KUKA KRL program: EPS_2_25730_SANMH01_A_20250909085214.src

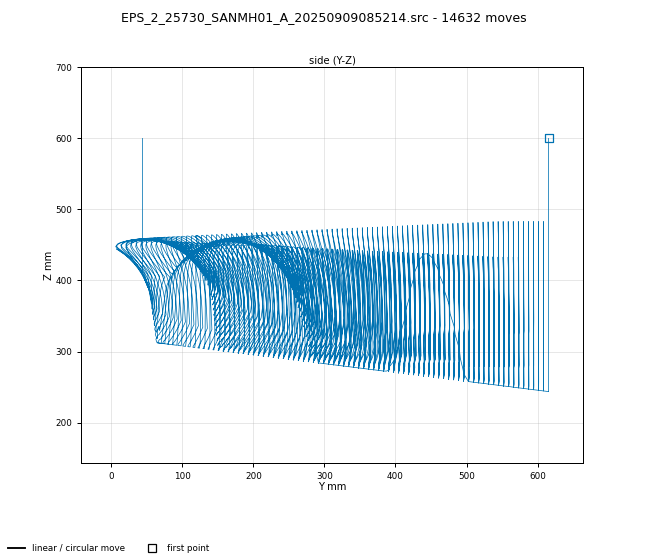
[picture p0: tool path of EPS_2_25730_SANMH01_A_20250909085214.src, 14632 of 14634 moves have a stored position in this frame; points joined in program order, loops and branches not executed]
&ACCESS RVP
&REL 4
&COMMENT QRS 19112012
&PARAM EDITMASK = *
DEF PART()
EXT BAS (BAS_COMMAND :IN,REAL :IN )
INT I
BAS (#INITMOV,0 )

;KUKA QRS Post kuka4.cps  Date:22-06-2017 !

File_ID=2821

QRS_PRE_INIT()

;Init var - Until changes are made in qrs_pre_init
Outlet_Square_prg=0
Inlet_1_Square_prg=0
Inlet_2_Square_prg=0
Inlet_3_Square_prg=0
Inlet_4_Square_prg=0
Inlet_5_Square_prg=0

Outlet_1={X 0.000, Y 541.230, Z 408.000, B 0.000, E1 0.000 }
Inlet_1={X 0.000, Y 544.780, Z 358.000, B 0.000, E1 163.000 }
Inlet_2={X 0.000, Y 544.780, Z 358.000, B 0.000, E1 270.000 }
Outlet_1_type=150
Inlet_1_type=150
Inlet_2_type=150
;QRS#1=Sidecore dimensions
;QRS#2=150-6" PVC SDR 28
;QRS#3=150-6" PVC SDR 28
;QRS#4=150-6" PVC SDR 28
;QRS#5=
;QRS#6=
;QRS#7=
;QRS#8=
;QRS#9=10-06 PSX
;QRS#10=10-06 PSX
;QRS#11=10-06 PSX
;QRS#12=
;QRS#13=
;QRS#14=
;QRS#15=
;QRS#16=1220x127x762 2,5'
;QRS#17=EPS Height
;QRS#18=483
;QRS#19=*
;QRS#20= UPDATED VERSION 22-06-2017
;QRS#21=*
Outlet_Square=070
Inlet_1_Square=070
Inlet_2_Square=070
Inlet_3_Square=0
Inlet_4_Square=0
Inlet_5_Square=0
Mill_Square=1
Outlet_Square_Prg=203
Inlet_1_Square_prg=203
Inlet_2_Square_prg=203

QRS_INIT()

$ADVANCE=5

; T1
PTP {E1 173.628,E2 173.628}
PTP {X 0,Y 615.477,A -85,B 0,C 180,E1 173.628,E2 173.628,E3 0,E4 0,E5 0,E6 0}
QRS_SPEED_INIT()
LIN {X 0,Y 615.477,Z 600,A -85,B 0,C 180,E1 173.628,E2 173.628,E3 0,E4 0,E5 0,E6 0} C_VEL
LIN {X 0,Y 615.477,Z 253.689,A -85,B 0,C 180,E1 173.628,E2 173.628} C_VEL
LIN {X 0,Y 615.477,Z 245.508,A -85,B 0,C 180,E1 173.628,E2 173.628} C_VEL
LIN {X 0,Y 615.462,Z 243.508,A -85,B 0,C 180,E1 173.442,E2 173.442} C_VEL
LIN {X 0,Y 615.457,Z 243.501,A -85,B 0,C 180,E1 170.803,E2 170.803} C_VEL
LIN {X 0,Y 615.49,Z 243.501,A -85,B 0,C 180,E1 168.142,E2 168.142} C_VEL
LIN {X 0,Y 615.471,Z 243.51,A -85,B 0,C 180,E1 165.453,E2 165.453} C_VEL
LIN {X 0,Y 615.469,Z 243.509,A -85,B 0,C 180,E1 163.416,E2 163.416} C_VEL
LIN {X 0,Y 615.466,Z 243.509,A -85,B 0,C 180,E1 161.356,E2 161.356} C_VEL
LIN {X 0,Y 615.462,Z 243.509,A -85,B 0,C 180,E1 159.271,E2 159.271} C_VEL
LIN {X 0,Y 615.456,Z 243.508,A -85,B 0,C 180,E1 157.157,E2 157.157} C_VEL
LIN {X 0,Y 615.45,Z 243.506,A -85,B 0,C 180,E1 155.01,E2 155.01} C_VEL
LIN {X 0,Y 615.446,Z 243.505,A -85,B 0,C 180,E1 152.824,E2 152.824} C_VEL
LIN {X 0,Y 615.475,Z 243.499,A -85,B 0,C 180,E1 150.207,E2 150.207} C_VEL
LIN {X 0,Y 615.493,Z 243.511,A -85,B 0,C 180,E1 147.547,E2 147.547} C_VEL
LIN {X 0,Y 615.469,Z 243.51,A -85,B 0,C 180,E1 145.188,E2 145.188} C_VEL
LIN {X 0,Y 615.444,Z 243.506,A -85,B 0,C 180,E1 142.759,E2 142.759} C_VEL
LIN {X 0,Y 615.489,Z 243.498,A -85,B 0,C 180,E1 139.911,E2 139.911} C_VEL
LIN {X 0,Y 615.458,Z 243.509,A -85,B 0,C 180,E1 136.956,E2 136.956} C_VEL
LIN {X 0,Y 615.458,Z 243.509,A -85,B 0,C 180,E1 134.934,E2 134.934} C_VEL
LIN {X 0,Y 615.443,Z 243.504,A -85,B 0,C 180,E1 132.357,E2 132.357} C_VEL
LIN {X 0,Y 615.488,Z 243.499,A -85,B 0,C 180,E1 129.75,E2 129.75} C_VEL
LIN {X 0,Y 615.467,Z 243.51,A -85,B 0,C 180,E1 126.94,E2 126.94} C_VEL
LIN {X 0,Y 615.45,Z 243.508,A -85,B 0,C 180,E1 124.702,E2 124.702} C_VEL
LIN {X 0,Y 615.49,Z 243.609,A -85,B 0,C 180,E1 123.602,E2 123.602} C_VEL
LIN {X 0,Y 615.443,Z 256.214,A -85,B 0,C 180,E1 120.922,E2 120.922} C_VEL
LIN {X 0,Y 615.478,Z 267.899,A -85,B 0,C 180,E1 118.457,E2 118.457} C_VEL
LIN {X 0,Y 615.482,Z 274.607,A -85,B 0,C 180,E1 117.053,E2 117.053} C_VEL
LIN {X 0,Y 615.469,Z 350.299,A -85,B 0,C 180,E1 116.148,E2 116.148} C_VEL
LIN {X 0,Y 615.466,Z 359.834,A -85,B 0,C 180,E1 115.944,E2 115.944} C_VEL
LIN {X 0,Y 615.476,Z 369.268,A -85,B 0,C 180,E1 115.647,E2 115.647} C_VEL
LIN {X 0,Y 615.495,Z 380.853,A -85,B 0,C 180,E1 115.137,E2 115.137} C_VEL
LIN {X 0,Y 615.481,Z 389.489,A -85,B 0,C 180,E1 114.632,E2 114.632} C_VEL
LIN {X 0,Y 615.487,Z 396.326,A -85,B 0,C 180,E1 114.145,E2 114.145} C_VEL
LIN {X 0,Y 615.497,Z 403.192,A -85,B 0,C 180,E1 113.556,E2 113.556} C_VEL
LIN {X 0,Y 615.495,Z 410.002,A -85,B 0,C 180,E1 112.844,E2 112.844} C_VEL
LIN {X 0,Y 615.496,Z 416.819,A -85,B 0,C 180,E1 111.96,E2 111.96} C_VEL
LIN {X 0,Y 615.497,Z 422.135,A -85,B 0,C 180,E1 111.08,E2 111.08} C_VEL
LIN {X 0,Y 615.492,Z 426.762,A -85,B 0,C 180,E1 110.033,E2 110.033} C_VEL
LIN {X 0,Y 615.495,Z 429.072,A -85,B 0,C 180,E1 109.338,E2 109.338} C_VEL
LIN {X 0,Y 615.489,Z 430.797,A -85,B 0,C 180,E1 108.618,E2 108.618} C_VEL
LIN {X 0,Y 615.489,Z 431.768,A -85,B 0,C 180,E1 107.957,E2 107.957} C_VEL
LIN {X 0,Y 615.498,Z 432.261,A -85,B 0,C 180,E1 107.27,E2 107.27} C_VEL
LIN {X 0,Y 615.494,Z 432.172,A -85,B 0,C 180,E1 106.448,E2 106.448} C_VEL
LIN {X 0,Y 615.492,Z 431.698,A -85,B 0,C 180,E1 105.905,E2 105.905} C_VEL
LIN {X 0,Y 615.496,Z 430.652,A -85,B 0,C 180,E1 105.226,E2 105.226} C_VEL
LIN {X 0,Y 615.495,Z 429.013,A -85,B 0,C 180,E1 104.549,E2 104.549} C_VEL
LIN {X 0,Y 615.49,Z 425.444,A -85,B 0,C 180,E1 103.537,E2 103.537} C_VEL
LIN {X 0,Y 615.495,Z 422.326,A -85,B 0,C 180,E1 102.865,E2 102.865} C_VEL
LIN {X 0,Y 615.495,Z 417.37,A -85,B 0,C 180,E1 102.028,E2 102.028} C_VEL
LIN {X 0,Y 615.5,Z 411.091,A -85,B 0,C 180,E1 101.193,E2 101.193} C_VEL
LIN {X 0,Y 615.498,Z 404.96,A -85,B 0,C 180,E1 100.527,E2 100.527} C_VEL
LIN {X 0,Y 615.494,Z 398.525,A -85,B 0,C 180,E1 99.945,E2 99.945} C_VEL
LIN {X 0,Y 615.489,Z 390.747,A -85,B 0,C 180,E1 99.364,E2 99.364} C_VEL
LIN {X 0,Y 615.486,Z 382.553,A -85,B 0,C 180,E1 98.867,E2 98.867} C_VEL
LIN {X 0,Y 615.442,Z 372.203,A -85,B 0,C 180,E1 98.372,E2 98.372} C_VEL
LIN {X 0,Y 615.439,Z 361.207,A -85,B 0,C 180,E1 98,E2 98} C_VEL
LIN {X 0,Y 615.451,Z 351.026,A -85,B 0,C 180,E1 97.773,E2 97.773} C_VEL
LIN {X 0,Y 615.489,Z 317.409,A -85,B 0,C 180,E1 97.36,E2 97.36} C_VEL
LIN {X 0,Y 615.47,Z 274.544,A -85,B 0,C 180,E1 96.843,E2 96.843} C_VEL
LIN {X 0,Y 615.484,Z 262.206,A -85,B 0,C 180,E1 94.256,E2 94.256} C_VEL
LIN {X 0,Y 615.456,Z 249.841,A -85,B 0,C 180,E1 91.636,E2 91.636} C_VEL
LIN {X 0,Y 615.44,Z 243.51,A -85,B 0,C 180,E1 90.245,E2 90.245} C_VEL
LIN {X 0,Y 615.428,Z 243.509,A -85,B 0,C 180,E1 88.037,E2 88.037} C_VEL
LIN {X 0,Y 615.429,Z 243.51,A -85,B 0,C 180,E1 86.071,E2 86.071} C_VEL
LIN {X 0,Y 615.43,Z 243.51,A -85,B 0,C 180,E1 84.101,E2 84.101} C_VEL
LIN {X 0,Y 615.432,Z 243.51,A -85,B 0,C 180,E1 82.124,E2 82.124} C_VEL
LIN {X 0,Y 615.433,Z 243.511,A -85,B 0,C 180,E1 80.137,E2 80.137} C_VEL
LIN {X 0,Y 615.433,Z 243.511,A -85,B 0,C 180,E1 78.138,E2 78.138} C_VEL
LIN {X 0,Y 615.429,Z 243.511,A -85,B 0,C 180,E1 76.072,E2 76.072} C_VEL
LIN {X 0,Y 615.431,Z 243.511,A -85,B 0,C 180,E1 74.093,E2 74.093} C_VEL
LIN {X 0,Y 615.428,Z 243.512,A -85,B 0,C 180,E1 72.041,E2 72.041} C_VEL
LIN {X 0,Y 615.423,Z 243.512,A -85,B 0,C 180,E1 69.965,E2 69.965} C_VEL
LIN {X 0,Y 615.41,Z 243.512,A -85,B 0,C 180,E1 67.661,E2 67.661} C_VEL
LIN {X 0,Y 615.411,Z 243.512,A -85,B 0,C 180,E1 65.725,E2 65.725} C_VEL
LIN {X 0,Y 615.407,Z 243.512,A -85,B 0,C 180,E1 63.552,E2 63.552} C_VEL
LIN {X 0,Y 615.486,Z 243.513,A -85,B 0,C 180,E1 60.593,E2 60.593} C_VEL
LIN {X 0,Y 615.411,Z 243.512,A -85,B 0,C 180,E1 57.673,E2 57.673} C_VEL
LIN {X 0,Y 615.435,Z 243.511,A -85,B 0,C 180,E1 55.974,E2 55.974} C_VEL
LIN {X 0,Y 615.413,Z 243.511,A -85,B 0,C 180,E1 53.57,E2 53.57} C_VEL
LIN {X 0,Y 615.428,Z 243.513,A -85,B 0,C 180,E1 50.939,E2 50.939} C_VEL
LIN {X 0,Y 615.479,Z 243.513,A -85,B 0,C 180,E1 48.525,E2 48.525} C_VEL
LIN {X 0,Y 615.442,Z 243.509,A -85,B 0,C 180,E1 45.846,E2 45.846} C_VEL
LIN {X 0,Y 615.463,Z 243.508,A -85,B 0,C 180,E1 43.995,E2 43.995} C_VEL
LIN {X 0,Y 615.424,Z 243.509,A -85,B 0,C 180,E1 41.474,E2 41.474} C_VEL
LIN {X 0,Y 615.425,Z 243.51,A -85,B 0,C 180,E1 39.055,E2 39.055} C_VEL
LIN {X 0,Y 615.477,Z 243.514,A -85,B 0,C 180,E1 36.421,E2 36.421} C_VEL
LIN {X 0,Y 615.436,Z 243.507,A -85,B 0,C 180,E1 33.527,E2 33.527} C_VEL
LIN {X 0,Y 615.428,Z 243.508,A -85,B 0,C 180,E1 31.076,E2 31.076} C_VEL
LIN {X 0,Y 615.445,Z 243.511,A -85,B 0,C 180,E1 28.657,E2 28.657} C_VEL
LIN {X 0,Y 615.47,Z 243.503,A -85,B 0,C 180,E1 25.713,E2 25.713} C_VEL
LIN {X 0,Y 615.457,Z 243.503,A -85,B 0,C 180,E1 23.554,E2 23.554} C_VEL
LIN {X 0,Y 615.45,Z 243.504,A -85,B 0,C 180,E1 21.43,E2 21.43} C_VEL
LIN {X 0,Y 615.446,Z 243.504,A -85,B 0,C 180,E1 19.336,E2 19.336} C_VEL
LIN {X 0,Y 615.437,Z 243.506,A -85,B 0,C 180,E1 16.927,E2 16.927} C_VEL
LIN {X 0,Y 615.451,Z 243.701,A -85,B 0,C 180,E1 16.585,E2 16.585} C_VEL
LIN {X 0,Y 615.492,Z 256.442,A -85,B 0,C 180,E1 13.871,E2 13.871} C_VEL
LIN {X 0,Y 615.492,Z 269.166,A -85,B 0,C 180,E1 11.19,E2 11.19} C_VEL
LIN {X 0,Y 615.458,Z 274.778,A -85,B 0,C 180,E1 10.047,E2 10.047} C_VEL
LIN {X 0,Y 615.452,Z 349.885,A -85,B 0,C 180,E1 9.155,E2 9.155} C_VEL
LIN {X 0,Y 615.441,Z 359.665,A -85,B 0,C 180,E1 8.949,E2 8.949} C_VEL
LIN {X 0,Y 615.439,Z 370.133,A -85,B 0,C 180,E1 8.618,E2 8.618} C_VEL
LIN {X 0,Y 615.476,Z 381.152,A -85,B 0,C 180,E1 8.121,E2 8.121} C_VEL
LIN {X 0,Y 615.494,Z 389.572,A -85,B 0,C 180,E1 7.626,E2 7.626} C_VEL
LIN {X 0,Y 615.493,Z 397.414,A -85,B 0,C 180,E1 7.056,E2 7.056} C_VEL
LIN {X 0,Y 615.498,Z 403.209,A -85,B 0,C 180,E1 6.554,E2 6.554} C_VEL
LIN {X 0,Y 615.499,Z 409.555,A -85,B 0,C 180,E1 5.896,E2 5.896} C_VEL
LIN {X 0,Y 615.495,Z 416,A -85,B 0,C 180,E1 5.075,E2 5.075} C_VEL
LIN {X 0,Y 615.492,Z 421.136,A -85,B 0,C 180,E1 4.254,E2 4.254} C_VEL
LIN {X 0,Y 615.494,Z 425.896,A -85,B 0,C 180,E1 3.271,E2 3.271} C_VEL
LIN {X 0,Y 615.493,Z 428.208,A -85,B 0,C 180,E1 2.616,E2 2.616} C_VEL
LIN {X 0,Y 615.494,Z 429.982,A -85,B 0,C 180,E1 1.961,E2 1.961} C_VEL
LIN {X 0,Y 615.496,Z 431.268,A -85,B 0,C 180,E1 1.306,E2 1.306} C_VEL
LIN {X 0,Y 615.491,Z 432.085,A -85,B 0,C 180,E1 0.652,E2 0.652} C_VEL
LIN {X 0,Y 615.492,Z 432.385,A -85,B 0,C 180,E1 -0.002,E2 -0.002} C_VEL
LIN {X 0,Y 615.494,Z 432.123,A -85,B 0,C 180,E1 -0.656,E2 -0.656} C_VEL
LIN {X 0,Y 615.494,Z 431.391,A -85,B 0,C 180,E1 -1.311,E2 -1.311} C_VEL
LIN {X 0,Y 615.497,Z 430.19,A -85,B 0,C 180,E1 -1.965,E2 -1.965} C_VEL
LIN {X 0,Y 615.49,Z 427.369,A -85,B 0,C 180,E1 -2.947,E2 -2.947} C_VEL
LIN {X 0,Y 615.49,Z 424.801,A -85,B 0,C 180,E1 -3.603,E2 -3.603} C_VEL
LIN {X 0,Y 615.498,Z 419.731,A -85,B 0,C 180,E1 -4.586,E2 -4.586} C_VEL
LIN {X 0,Y 615.496,Z 414.274,A -85,B 0,C 180,E1 -5.407,E2 -5.407} C_VEL
LIN {X 0,Y 615.497,Z 407.435,A -85,B 0,C 180,E1 -6.229,E2 -6.229} C_VEL
LIN {X 0,Y 615.497,Z 400.414,A -85,B 0,C 180,E1 -6.901,E2 -6.901} C_VEL
LIN {X 0,Y 615.478,Z 392.046,A -85,B 0,C 180,E1 -7.547,E2 -7.547} C_VEL
LIN {X 0,Y 615.497,Z 384.162,A -85,B 0,C 180,E1 -8.042,E2 -8.042} C_VEL
LIN {X 0,Y 615.492,Z 376.033,A -85,B 0,C 180,E1 -8.456,E2 -8.456} C_VEL
LIN {X 0,Y 615.486,Z 367.81,A -85,B 0,C 180,E1 -8.787,E2 -8.787} C_VEL
LIN {X 0,Y 615.475,Z 359.771,A -85,B 0,C 180,E1 -9.035,E2 -9.035} C_VEL
LIN {X 0,Y 615.475,Z 350.054,A -85,B 0,C 180,E1 -9.242,E2 -9.242} C_VEL
LIN {X 0,Y 615.477,Z 274.551,A -85,B 0,C 180,E1 -10.155,E2 -10.155} C_VEL
LIN {X 0,Y 615.496,Z 261.617,A -85,B 0,C 180,E1 -12.867,E2 -12.867} C_VEL
LIN {X 0,Y 615.447,Z 248.888,A -85,B 0,C 180,E1 -15.568,E2 -15.568} C_VEL
LIN {X 0,Y 615.488,Z 243.499,A -85,B 0,C 180,E1 -16.759,E2 -16.759} C_VEL
LIN {X 0,Y 615.454,Z 243.502,A -85,B 0,C 180,E1 -19.341,E2 -19.341} C_VEL
LIN {X 0,Y 615.452,Z 243.502,A -85,B 0,C 180,E1 -21.435,E2 -21.435} C_VEL
LIN {X 0,Y 615.466,Z 243.509,A -85,B 0,C 180,E1 -24.003,E2 -24.003} C_VEL
LIN {X 0,Y 615.496,Z 243.51,A -85,B 0,C 180,E1 -26.445,E2 -26.445} C_VEL
LIN {X 0,Y 615.491,Z 243.504,A -85,B 0,C 180,E1 -28.659,E2 -28.659} C_VEL
LIN {X 0,Y 615.481,Z 243.497,A -85,B 0,C 180,E1 -31.085,E2 -31.085} C_VEL
LIN {X 0,Y 615.459,Z 243.5,A -85,B 0,C 180,E1 -33.53,E2 -33.53} C_VEL
LIN {X 0,Y 615.456,Z 243.504,A -85,B 0,C 180,E1 -35.829,E2 -35.829} C_VEL
LIN {X 0,Y 615.463,Z 243.507,A -85,B 0,C 180,E1 -38.071,E2 -38.071} C_VEL
LIN {X 0,Y 615.495,Z 243.51,A -85,B 0,C 180,E1 -40.607,E2 -40.607} C_VEL
LIN {X 0,Y 615.497,Z 243.493,A -85,B 0,C 180,E1 -43.245,E2 -43.245} C_VEL
LIN {X 0,Y 615.46,Z 243.504,A -85,B 0,C 180,E1 -46.006,E2 -46.006} C_VEL
LIN {X 0,Y 615.488,Z 243.504,A -85,B 0,C 180,E1 -48.906,E2 -48.906} C_VEL
LIN {X 0,Y 615.487,Z 243.5,A -85,B 0,C 180,E1 -51.095,E2 -51.095} C_VEL
LIN {X 0,Y 615.478,Z 243.496,A -85,B 0,C 180,E1 -53.574,E2 -53.574} C_VEL
LIN {X 0,Y 615.462,Z 243.501,A -85,B 0,C 180,E1 -55.976,E2 -55.976} C_VEL
LIN {X 0,Y 615.465,Z 243.507,A -85,B 0,C 180,E1 -58.313,E2 -58.313} C_VEL
LIN {X 0,Y 615.481,Z 243.511,A -85,B 0,C 180,E1 -60.593,E2 -60.593} C_VEL
LIN {X 0,Y 615.491,Z 243.494,A -85,B 0,C 180,E1 -63.556,E2 -63.556} C_VEL
LIN {X 0,Y 615.47,Z 243.499,A -85,B 0,C 180,E1 -65.996,E2 -65.996} C_VEL
LIN {X 0,Y 615.467,Z 243.585,A -85,B 0,C 180,E1 -68.193,E2 -68.193} C_VEL
LIN {X 0,Y 615.47,Z 260.981,A -85,B 0,C 180,E1 -70.835,E2 -70.835} C_VEL
LIN {X 0,Y 615.46,Z 278.212,A -85,B 0,C 180,E1 -73.412,E2 -73.412} C_VEL
LIN {X 0,Y 615.461,Z 297.724,A -85,B 0,C 180,E1 -76.293,E2 -76.293} C_VEL
LIN {X 0,Y 615.48,Z 316,A -85,B 0,C 180,E1 -78.963,E2 -78.963} C_VEL
LIN {X 0,Y 615.498,Z 322.219,A -85,B 0,C 180,E1 -79.868,E2 -79.868} C_VEL
LIN {X 0,Y 615.457,Z 399.942,A -85,B 0,C 180,E1 -80.801,E2 -80.801} C_VEL
LIN {X 0,Y 615.449,Z 409.702,A -85,B 0,C 180,E1 -81.008,E2 -81.008} C_VEL
LIN {X 0,Y 615.452,Z 420.16,A -85,B 0,C 180,E1 -81.339,E2 -81.339} C_VEL
LIN {X 0,Y 615.484,Z 430.427,A -85,B 0,C 180,E1 -81.794,E2 -81.794} C_VEL
LIN {X 0,Y 615.478,Z 440.199,A -85,B 0,C 180,E1 -82.372,E2 -82.372} C_VEL
LIN {X 0,Y 615.493,Z 447.935,A -85,B 0,C 180,E1 -82.942,E2 -82.942} C_VEL
LIN {X 0,Y 615.498,Z 455.332,A -85,B 0,C 180,E1 -83.608,E2 -83.608} C_VEL
LIN {X 0,Y 615.498,Z 462.736,A -85,B 0,C 180,E1 -84.43,E2 -84.43} C_VEL
LIN {X 0,Y 615.497,Z 468.532,A -85,B 0,C 180,E1 -85.251,E2 -85.251} C_VEL
LIN {X 0,Y 615.496,Z 473.099,A -85,B 0,C 180,E1 -86.071,E2 -86.071} C_VEL
LIN {X 0,Y 615.493,Z 476.068,A -85,B 0,C 180,E1 -86.727,E2 -86.727} C_VEL
LIN {X 0,Y 615.494,Z 478.356,A -85,B 0,C 180,E1 -87.382,E2 -87.382} C_VEL
LIN {X 0,Y 615.499,Z 480.085,A -85,B 0,C 180,E1 -88.037,E2 -88.037} C_VEL
LIN {X 0,Y 615.493,Z 481.33,A -85,B 0,C 180,E1 -88.691,E2 -88.691} C_VEL
LIN {X 0,Y 615.491,Z 482.104,A -85,B 0,C 180,E1 -89.346,E2 -89.346} C_VEL
LIN {X 0,Y 615.491,Z 482.389,A -85,B 0,C 180,E1 -90,E2 -90} C_VEL
LIN {X 0,Y 615.491,Z 482.104,A -85,B 0,C 180,E1 -90.654,E2 -90.654} C_VEL
LIN {X 0,Y 615.493,Z 481.33,A -85,B 0,C 180,E1 -91.308,E2 -91.308} C_VEL
LIN {X 0,Y 615.499,Z 480.085,A -85,B 0,C 180,E1 -91.963,E2 -91.963} C_VEL
LIN {X 0,Y 615.488,Z 477.221,A -85,B 0,C 180,E1 -92.945,E2 -92.945} C_VEL
LIN {X 0,Y 615.493,Z 474.603,A -85,B 0,C 180,E1 -93.601,E2 -93.601} C_VEL
LIN {X 0,Y 615.496,Z 469.483,A -85,B 0,C 180,E1 -94.584,E2 -94.584} C_VEL
LIN {X 0,Y 615.495,Z 463.969,A -85,B 0,C 180,E1 -95.405,E2 -95.405} C_VEL
LIN {X 0,Y 615.499,Z 457.019,A -85,B 0,C 180,E1 -96.227,E2 -96.227} C_VEL
LIN {X 0,Y 615.495,Z 449.862,A -85,B 0,C 180,E1 -96.901,E2 -96.901} C_VEL
LIN {X 0,Y 615.477,Z 442.626,A -85,B 0,C 180,E1 -97.463,E2 -97.463} C_VEL
LIN {X 0,Y 615.495,Z 434.87,A -85,B 0,C 180,E1 -97.958,E2 -97.958} C_VEL
LIN {X 0,Y 615.473,Z 426.922,A -85,B 0,C 180,E1 -98.371,E2 -98.371} C_VEL
LIN {X 0,Y 615.45,Z 417.771,A -85,B 0,C 180,E1 -98.744,E2 -98.744} C_VEL
LIN {X 0,Y 615.449,Z 409.713,A -85,B 0,C 180,E1 -98.992,E2 -98.992} C_VEL
LIN {X 0,Y 615.457,Z 399.959,A -85,B 0,C 180,E1 -99.199,E2 -99.199} C_VEL
LIN {X 0,Y 615.498,Z 322.221,A -85,B 0,C 180,E1 -100.132,E2 -100.132} C_VEL
LIN {X 0,Y 615.486,Z 302.31,A -85,B 0,C 180,E1 -103.033,E2 -103.033} C_VEL
LIN {X 0,Y 615.437,Z 285.108,A -85,B 0,C 180,E1 -105.567,E2 -105.567} C_VEL
LIN {X 0,Y 615.484,Z 265.807,A -85,B 0,C 180,E1 -108.439,E2 -108.439} C_VEL
LIN {X 0,Y 615.486,Z 247.181,A -85,B 0,C 180,E1 -111.256,E2 -111.256} C_VEL
LIN {X 0,Y 615.466,Z 243.501,A -85,B 0,C 180,E1 -111.828,E2 -111.828} C_VEL
LIN {X 0,Y 615.487,Z 243.494,A -85,B 0,C 180,E1 -114.272,E2 -114.272} C_VEL
LIN {X 0,Y 615.485,Z 243.513,A -85,B 0,C 180,E1 -117.177,E2 -117.177} C_VEL
LIN {X 0,Y 615.466,Z 243.504,A -85,B 0,C 180,E1 -119.791,E2 -119.791} C_VEL
LIN {X 0,Y 615.487,Z 243.494,A -85,B 0,C 180,E1 -122.457,E2 -122.457} C_VEL
LIN {X 0,Y 615.488,Z 243.498,A -85,B 0,C 180,E1 -124.815,E2 -124.815} C_VEL
LIN {X 0,Y 615.488,Z 243.509,A -85,B 0,C 180,E1 -127.242,E2 -127.242} C_VEL
LIN {X 0,Y 615.463,Z 243.502,A -85,B 0,C 180,E1 -130.086,E2 -130.086} C_VEL
LIN {X 0,Y 615.47,Z 243.498,A -85,B 0,C 180,E1 -132.354,E2 -132.354} C_VEL
LIN {X 0,Y 615.487,Z 243.501,A -85,B 0,C 180,E1 -135.069,E2 -135.069} C_VEL
LIN {X 0,Y 615.487,Z 243.511,A -85,B 0,C 180,E1 -137.646,E2 -137.646} C_VEL
LIN {X 0,Y 615.461,Z 243.502,A -85,B 0,C 180,E1 -140.247,E2 -140.247} C_VEL
LIN {X 0,Y 615.491,Z 243.498,A -85,B 0,C 180,E1 -143.063,E2 -143.063} C_VEL
LIN {X 0,Y 615.469,Z 243.507,A -85,B 0,C 180,E1 -145.976,E2 -145.976} C_VEL
LIN {X 0,Y 615.46,Z 243.503,A -85,B 0,C 180,E1 -148.312,E2 -148.312} C_VEL
LIN {X 0,Y 615.464,Z 243.499,A -85,B 0,C 180,E1 -150.591,E2 -150.591} C_VEL
LIN {X 0,Y 615.49,Z 243.508,A -85,B 0,C 180,E1 -153.555,E2 -153.555} C_VEL
LIN {X 0,Y 615.477,Z 243.509,A -85,B 0,C 180,E1 -155.994,E2 -155.994} C_VEL
LIN {X 0,Y 615.458,Z 243.502,A -85,B 0,C 180,E1 -158.566,E2 -158.566} C_VEL
LIN {X 0,Y 615.489,Z 243.5,A -85,B 0,C 180,E1 -161.395,E2 -161.395} C_VEL
LIN {X 0,Y 615.477,Z 243.51,A -85,B 0,C 180,E1 -164.093,E2 -164.093} C_VEL
LIN {X 0,Y 615.459,Z 243.5,A -85,B 0,C 180,E1 -166.796,E2 -166.796} C_VEL
LIN {X 0,Y 615.49,Z 243.499,A -85,B 0,C 180,E1 -169.471,E2 -169.471} C_VEL
LIN {X 0,Y 615.484,Z 243.511,A -85,B 0,C 180,E1 -172.123,E2 -172.123} C_VEL
LIN {X 0,Y 615.452,Z 243.503,A -85,B 0,C 180,E1 -174.757,E2 -174.757} C_VEL
LIN {X 0,Y 615.491,Z 243.495,A -85,B 0,C 180,E1 -177.38,E2 -177.38} C_VEL
LIN {X 0,Y 615.488,Z 243.511,A -85,B 0,C 180,E1 -179.998,E2 -179.998} C_VEL
LIN {X 0,Y 615.457,Z 243.506,A -85,B 0,C 180,E1 -182.616,E2 -182.616} C_VEL
LIN {X 0,Y 615.464,Z 243.499,A -85,B 0,C 180,E1 -185.239,E2 -185.239} C_VEL
LIN {X 0,Y 615.462,Z 243.508,A -85,B 0,C 180,E1 -186.558,E2 -186.558} C_VEL
LIN {X 0,Y 614.783,Z 243.648,A -85,B 0,C 180,E1 -187.104,E2 -187.104} C_VEL
LIN {X 0,Y 611.943,Z 244.072,A -85,B 0,C 180,E1 -187.99,E2 -187.99} C_VEL
LIN {X 0,Y 609.554,Z 244.377,A -85,B 0,C 180,E1 -188.702,E2 -188.702} C_VEL
LIN {X 0,Y 608.528,Z 244.491,A -85,B 0,C 180,E1 -189.252,E2 -189.252} C_VEL
LIN {X 0,Y 608.444,Z 244.501,A -85,B 0,C 180,E1 -189.438,E2 -189.438} C_VEL
LIN {X 0,Y 608.461,Z 244.505,A -85,B 0,C 180,E1 -191.997,E2 -191.997} C_VEL
LIN {X 0,Y 608.457,Z 244.502,A -85,B 0,C 180,E1 -194.718,E2 -194.718} C_VEL
LIN {X 0,Y 608.434,Z 244.502,A -85,B 0,C 180,E1 -197.474,E2 -197.474} C_VEL
LIN {X 0,Y 608.462,Z 244.508,A -85,B 0,C 180,E1 -200.271,E2 -200.271} C_VEL
LIN {X 0,Y 608.425,Z 244.503,A -85,B 0,C 180,E1 -203.122,E2 -203.122} C_VEL
LIN {X 0,Y 608.455,Z 244.5,A -85,B 0,C 180,E1 -205.718,E2 -205.718} C_VEL
LIN {X 0,Y 608.469,Z 244.506,A -85,B 0,C 180,E1 -208.619,E2 -208.619} C_VEL
LIN {X 0,Y 608.423,Z 244.503,A -85,B 0,C 180,E1 -211.315,E2 -211.315} C_VEL
LIN {X 0,Y 608.453,Z 244.5,A -85,B 0,C 180,E1 -213.732,E2 -213.732} C_VEL
LIN {X 0,Y 608.461,Z 244.501,A -85,B 0,C 180,E1 -216.087,E2 -216.087} C_VEL
LIN {X 0,Y 608.455,Z 244.51,A -85,B 0,C 180,E1 -218.585,E2 -218.585} C_VEL
LIN {X 0,Y 608.424,Z 244.504,A -85,B 0,C 180,E1 -221.338,E2 -221.338} C_VEL
LIN {X 0,Y 608.451,Z 244.5,A -85,B 0,C 180,E1 -223.866,E2 -223.866} C_VEL
LIN {X 0,Y 608.477,Z 244.507,A -85,B 0,C 180,E1 -226.685,E2 -226.685} C_VEL
LIN {X 0,Y 608.449,Z 244.51,A -85,B 0,C 180,E1 -228.823,E2 -228.823} C_VEL
LIN {X 0,Y 608.441,Z 244.502,A -85,B 0,C 180,E1 -231.41,E2 -231.41} C_VEL
LIN {X 0,Y 608.448,Z 244.5,A -85,B 0,C 180,E1 -233.948,E2 -233.948} C_VEL
LIN {X 0,Y 608.464,Z 244.6,A -85,B 0,C 180,E1 -236.379,E2 -236.379} C_VEL
LIN {X 0,Y 608.407,Z 257.241,A -85,B 0,C 180,E1 -239.088,E2 -239.088} C_VEL
LIN {X 0,Y 608.443,Z 269.722,A -85,B 0,C 180,E1 -241.733,E2 -241.733} C_VEL
LIN {X 0,Y 608.445,Z 274.939,A -85,B 0,C 180,E1 -242.831,E2 -242.831} C_VEL
LIN {X 0,Y 608.485,Z 350.231,A -85,B 0,C 180,E1 -243.736,E2 -243.736} C_VEL
LIN {X 0,Y 608.483,Z 359.852,A -85,B 0,C 180,E1 -243.943,E2 -243.943} C_VEL
LIN {X 0,Y 608.495,Z 370.84,A -85,B 0,C 180,E1 -244.296,E2 -244.296} C_VEL
LIN {X 0,Y 608.479,Z 381.599,A -85,B 0,C 180,E1 -244.792,E2 -244.792} C_VEL
LIN {X 0,Y 608.46,Z 390.688,A -85,B 0,C 180,E1 -245.338,E2 -245.338} C_VEL
LIN {X 0,Y 608.45,Z 397.565,A -85,B 0,C 180,E1 -245.843,E2 -245.843} C_VEL
LIN {X 0,Y 608.452,Z 405.104,A -85,B 0,C 180,E1 -246.516,E2 -246.516} C_VEL
LIN {X 0,Y 608.459,Z 411.693,A -85,B 0,C 180,E1 -247.234,E2 -247.234} C_VEL
LIN {X 0,Y 608.451,Z 418.332,A -85,B 0,C 180,E1 -248.13,E2 -248.13} C_VEL
LIN {X 0,Y 608.458,Z 423.391,A -85,B 0,C 180,E1 -249.019,E2 -249.019} C_VEL
LIN {X 0,Y 608.438,Z 426.586,A -85,B 0,C 180,E1 -249.725,E2 -249.725} C_VEL
LIN {X 0,Y 608.424,Z 429.041,A -85,B 0,C 180,E1 -250.429,E2 -250.429} C_VEL
LIN {X 0,Y 608.416,Z 431.227,A -85,B 0,C 180,E1 -251.287,E2 -251.287} C_VEL
LIN {X 0,Y 608.418,Z 432.779,A -85,B 0,C 180,E1 -252.523,E2 -252.523} C_VEL
LIN {X 0,Y 608.419,Z 432.824,A -85,B 0,C 180,E1 -253.472,E2 -253.472} C_VEL
LIN {X 0,Y 608.448,Z 432.578,A -85,B 0,C 180,E1 -253.906,E2 -253.906} C_VEL
LIN {X 0,Y 608.419,Z 431.616,A -85,B 0,C 180,E1 -254.593,E2 -254.593} C_VEL
LIN {X 0,Y 608.424,Z 429.181,A -85,B 0,C 180,E1 -255.62,E2 -255.62} C_VEL
LIN {X 0,Y 608.44,Z 425.348,A -85,B 0,C 180,E1 -256.643,E2 -256.643} C_VEL
LIN {X 0,Y 608.453,Z 420.106,A -85,B 0,C 180,E1 -257.662,E2 -257.662} C_VEL
LIN {X 0,Y 608.46,Z 414.471,A -85,B 0,C 180,E1 -258.507,E2 -258.507} C_VEL
LIN {X 0,Y 608.448,Z 407.387,A -85,B 0,C 180,E1 -259.35,E2 -259.35} C_VEL
LIN {X 0,Y 608.452,Z 399.265,A -85,B 0,C 180,E1 -260.107,E2 -260.107} C_VEL
LIN {X 0,Y 608.476,Z 391.52,A -85,B 0,C 180,E1 -260.694,E2 -260.694} C_VEL
LIN {X 0,Y 608.463,Z 383.406,A -85,B 0,C 180,E1 -261.197,E2 -261.197} C_VEL
LIN {X 0,Y 608.439,Z 373.155,A -85,B 0,C 180,E1 -261.698,E2 -261.698} C_VEL
LIN {X 0,Y 608.461,Z 361.063,A -85,B 0,C 180,E1 -262.116,E2 -262.116} C_VEL
LIN {X 0,Y 608.464,Z 350.74,A -85,B 0,C 180,E1 -262.346,E2 -262.346} C_VEL
LIN {X 0,Y 608.526,Z 311.68,A -85,B 0,C 180,E1 -262.825,E2 -262.825} C_VEL
LIN {X 0,Y 608.428,Z 274.911,A -85,B 0,C 180,E1 -263.265,E2 -263.265} C_VEL
LIN {X 0,Y 608.44,Z 261.83,A -85,B 0,C 180,E1 -266.026,E2 -266.026} C_VEL
LIN {X 0,Y 608.452,Z 249.408,A -85,B 0,C 180,E1 -268.676,E2 -268.676} C_VEL
LIN {X 0,Y 608.411,Z 244.507,A -85,B 0,C 180,E1 -269.752,E2 -269.752} C_VEL
LIN {X 0,Y 608.399,Z 244.507,A -85,B 0,C 180,E1 -271.986,E2 -271.986} C_VEL
LIN {X 0,Y 608.399,Z 244.507,A -85,B 0,C 180,E1 -273.974,E2 -273.974} C_VEL
LIN {X 0,Y 608.404,Z 244.507,A -85,B 0,C 180,E1 -275.968,E2 -275.968} C_VEL
LIN {X 0,Y 608.425,Z 244.504,A -85,B 0,C 180,E1 -277.968,E2 -277.968} C_VEL
LIN {X 0,Y 608.402,Z 244.507,A -85,B 0,C 180,E1 -279.978,E2 -279.978} C_VEL
LIN {X 0,Y 608.408,Z 244.506,A -85,B 0,C 180,E1 -282.001,E2 -282.001} C_VEL
LIN {X 0,Y 608.404,Z 244.506,A -85,B 0,C 180,E1 -284.039,E2 -284.039} C_VEL
LIN {X 0,Y 608.411,Z 244.505,A -85,B 0,C 180,E1 -286.525,E2 -286.525} C_VEL
LIN {X 0,Y 608.414,Z 244.507,A -85,B 0,C 180,E1 -288.871,E2 -288.871} C_VEL
LIN {X 0,Y 608.445,Z 244.506,A -85,B 0,C 180,E1 -291.693,E2 -291.693} C_VEL
LIN {X 0,Y 608.394,Z 244.507,A -85,B 0,C 180,E1 -294.574,E2 -294.574} C_VEL
LIN {X 0,Y 608.445,Z 244.507,A -85,B 0,C 180,E1 -297.21,E2 -297.21} C_VEL
LIN {X 0,Y 608.403,Z 244.509,A -85,B 0,C 180,E1 -299.969,E2 -299.969} C_VEL
LIN {X 0,Y 608.391,Z 244.507,A -85,B 0,C 180,E1 -302.519,E2 -302.519} C_VEL
LIN {X 0,Y 608.405,Z 244.505,A -85,B 0,C 180,E1 -304.474,E2 -304.474} C_VEL
LIN {X 0,Y 608.434,Z 244.506,A -85,B 0,C 180,E1 -307.16,E2 -307.16} C_VEL
LIN {X 0,Y 608.421,Z 244.512,A -85,B 0,C 180,E1 -309.444,E2 -309.444} C_VEL
LIN {X 0,Y 608.425,Z 244.506,A -85,B 0,C 180,E1 -312.065,E2 -312.065} C_VEL
LIN {X 0,Y 608.398,Z 244.506,A -85,B 0,C 180,E1 -314.802,E2 -314.802} C_VEL
LIN {X 0,Y 608.398,Z 244.508,A -85,B 0,C 180,E1 -317.04,E2 -317.04} C_VEL
LIN {X 0,Y 608.443,Z 244.511,A -85,B 0,C 180,E1 -319.7,E2 -319.7} C_VEL
LIN {X 0,Y 608.442,Z 244.503,A -85,B 0,C 180,E1 -322.256,E2 -322.256} C_VEL
LIN {X 0,Y 608.4,Z 244.506,A -85,B 0,C 180,E1 -324.724,E2 -324.724} C_VEL
LIN {X 0,Y 608.445,Z 244.507,A -85,B 0,C 180,E1 -327.481,E2 -327.481} C_VEL
LIN {X 0,Y 608.455,Z 244.502,A -85,B 0,C 180,E1 -330.223,E2 -330.223} C_VEL
LIN {X 0,Y 608.411,Z 244.505,A -85,B 0,C 180,E1 -332.806,E2 -332.806} C_VEL
LIN {X 0,Y 608.431,Z 244.507,A -85,B 0,C 180,E1 -335.431,E2 -335.431} C_VEL
LIN {X 0,Y 608.45,Z 244.502,A -85,B 0,C 180,E1 -338.311,E2 -338.311} C_VEL
LIN {X 0,Y 608.429,Z 244.503,A -85,B 0,C 180,E1 -341.133,E2 -341.133} C_VEL
LIN {X 0,Y 608.431,Z 244.708,A -85,B 0,C 180,E1 -343.402,E2 -343.402} C_VEL
LIN {X 0,Y 608.467,Z 258.302,A -85,B 0,C 180,E1 -346.315,E2 -346.315} C_VEL
LIN {X 0,Y 608.411,Z 271.344,A -85,B 0,C 180,E1 -349.074,E2 -349.074} C_VEL
LIN {X 0,Y 608.403,Z 274.864,A -85,B 0,C 180,E1 -349.814,E2 -349.814} C_VEL
LIN {X 0,Y 608.491,Z 343.22,A -85,B 0,C 180,E1 -350.634,E2 -350.634} C_VEL
LIN {X 0,Y 608.446,Z 355.921,A -85,B 0,C 180,E1 -350.843,E2 -350.843} C_VEL
LIN {X 0,Y 608.435,Z 365.683,A -85,B 0,C 180,E1 -351.115,E2 -351.115} C_VEL
LIN {X 0,Y 608.451,Z 374.456,A -85,B 0,C 180,E1 -351.45,E2 -351.45} C_VEL
LIN {X 0,Y 608.476,Z 382.971,A -85,B 0,C 180,E1 -351.868,E2 -351.868} C_VEL
LIN {X 0,Y 608.472,Z 391.145,A -85,B 0,C 180,E1 -352.369,E2 -352.369} C_VEL
LIN {X 0,Y 608.481,Z 398.902,A -85,B 0,C 180,E1 -352.953,E2 -352.953} C_VEL
LIN {X 0,Y 608.452,Z 407.012,A -85,B 0,C 180,E1 -353.703,E2 -353.703} C_VEL
LIN {X 0,Y 608.461,Z 414.126,A -85,B 0,C 180,E1 -354.534,E2 -354.534} C_VEL
LIN {X 0,Y 608.445,Z 419.738,A -85,B 0,C 180,E1 -355.365,E2 -355.365} C_VEL
LIN {X 0,Y 608.447,Z 424.951,A -85,B 0,C 180,E1 -356.36,E2 -356.36} C_VEL
LIN {X 0,Y 608.447,Z 427.639,A -85,B 0,C 180,E1 -357.023,E2 -357.023} C_VEL
LIN {X 0,Y 608.439,Z 430.576,A -85,B 0,C 180,E1 -358.016,E2 -358.016} C_VEL
LIN {X 0,Y 608.448,Z 431.874,A -85,B 0,C 180,E1 -358.678,E2 -358.678} C_VEL
LIN {X 0,Y 608.434,Z 432.695,A -85,B 0,C 180,E1 -359.34,E2 -359.34} C_VEL
LIN {X 0,Y 608.432,Z 432.995,A -85,B 0,C 180,E1 -360.002,E2 -360.002} C_VEL
LIN {X 0,Y 608.437,Z 432.736,A -85,B 0,C 180,E1 -360.664,E2 -360.664} C_VEL
LIN {X 0,Y 608.446,Z 431.996,A -85,B 0,C 180,E1 -361.326,E2 -361.326} C_VEL
LIN {X 0,Y 608.443,Z 430.783,A -85,B 0,C 180,E1 -361.988,E2 -361.988} C_VEL
LIN {X 0,Y 608.446,Z 427.935,A -85,B 0,C 180,E1 -362.982,E2 -362.982} C_VEL
LIN {X 0,Y 608.444,Z 425.343,A -85,B 0,C 180,E1 -363.644,E2 -363.644} C_VEL
LIN {X 0,Y 608.447,Z 420.233,A -85,B 0,C 180,E1 -364.64,E2 -364.64} C_VEL
LIN {X 0,Y 608.461,Z 414.735,A -85,B 0,C 180,E1 -365.47,E2 -365.47} C_VEL
LIN {X 0,Y 608.454,Z 407.165,A -85,B 0,C 180,E1 -366.372,E2 -366.372} C_VEL
LIN {X 0,Y 608.463,Z 398.931,A -85,B 0,C 180,E1 -367.135,E2 -367.135} C_VEL
LIN {X 0,Y 608.459,Z 391.178,A -85,B 0,C 180,E1 -367.719,E2 -367.719} C_VEL
LIN {X 0,Y 608.474,Z 383.009,A -85,B 0,C 180,E1 -368.219,E2 -368.219} C_VEL
LIN {X 0,Y 608.499,Z 372.645,A -85,B 0,C 180,E1 -368.721,E2 -368.721} C_VEL
LIN {X 0,Y 608.49,Z 360.977,A -85,B 0,C 180,E1 -369.119,E2 -369.119} C_VEL
LIN {X 0,Y 608.481,Z 350.543,A -85,B 0,C 180,E1 -369.349,E2 -369.349} C_VEL
LIN {X 0,Y 608.506,Z 284.345,A -85,B 0,C 180,E1 -370.146,E2 -370.146} C_VEL
LIN {X 0,Y 608.437,Z 274.871,A -85,B 0,C 180,E1 -370.274,E2 -370.274} C_VEL
LIN {X 0,Y 608.45,Z 261.865,A -85,B 0,C 180,E1 -373.019,E2 -373.019} C_VEL
LIN {X 0,Y 608.432,Z 249.058,A -85,B 0,C 180,E1 -375.752,E2 -375.752} C_VEL
LIN {X 0,Y 608.469,Z 244.5,A -85,B 0,C 180,E1 -376.74,E2 -376.74} C_VEL
LIN {X 0,Y 608.43,Z 244.503,A -85,B 0,C 180,E1 -379.573,E2 -379.573} C_VEL
LIN {X 0,Y 608.447,Z 244.502,A -85,B 0,C 180,E1 -381.694,E2 -381.694} C_VEL
LIN {X 0,Y 608.455,Z 244.506,A -85,B 0,C 180,E1 -384.572,E2 -384.572} C_VEL
LIN {X 0,Y 608.434,Z 244.502,A -85,B 0,C 180,E1 -387.52,E2 -387.52} C_VEL
LIN {X 0,Y 608.445,Z 244.504,A -85,B 0,C 180,E1 -389.967,E2 -389.967} C_VEL
LIN {X 0,Y 608.457,Z 244.502,A -85,B 0,C 180,E1 -392.881,E2 -392.881} C_VEL
LIN {X 0,Y 608.43,Z 244.502,A -85,B 0,C 180,E1 -395.28,E2 -395.28} C_VEL
LIN {X 0,Y 608.455,Z 244.5,A -85,B 0,C 180,E1 -397.748,E2 -397.748} C_VEL
LIN {X 0,Y 608.443,Z 244.508,A -85,B 0,C 180,E1 -400.328,E2 -400.328} C_VEL
LIN {X 0,Y 608.483,Z 244.496,A -85,B 0,C 180,E1 -403.31,E2 -403.31} C_VEL
LIN {X 0,Y 608.452,Z 244.503,A -85,B 0,C 180,E1 -406.129,E2 -406.129} C_VEL
LIN {X 0,Y 608.458,Z 244.506,A -85,B 0,C 180,E1 -408.823,E2 -408.823} C_VEL
LIN {X 0,Y 608.452,Z 244.5,A -85,B 0,C 180,E1 -411.762,E2 -411.762} C_VEL
LIN {X 0,Y 608.443,Z 244.501,A -85,B 0,C 180,E1 -413.956,E2 -413.956} C_VEL
LIN {X 0,Y 608.447,Z 244.505,A -85,B 0,C 180,E1 -416.328,E2 -416.328} C_VEL
LIN {X 0,Y 608.45,Z 244.511,A -85,B 0,C 180,E1 -418.733,E2 -418.733} C_VEL
LIN {X 0,Y 608.476,Z 244.498,A -85,B 0,C 180,E1 -421.38,E2 -421.38} C_VEL
LIN {X 0,Y 608.437,Z 244.502,A -85,B 0,C 180,E1 -423.964,E2 -423.964} C_VEL
LIN {X 0,Y 608.453,Z 244.501,A -85,B 0,C 180,E1 -426.154,E2 -426.154} C_VEL
LIN {X 0,Y 608.47,Z 244.6,A -85,B 0,C 180,E1 -428.086,E2 -428.086} C_VEL
LIN {X 0,Y 608.536,Z 259.861,A -85,B 0,C 180,E1 -430.432,E2 -430.432} C_VEL
LIN {X 0,Y 608.46,Z 277.136,A -85,B 0,C 180,E1 -433.043,E2 -433.043} C_VEL
LIN {X 0,Y 608.479,Z 296.831,A -85,B 0,C 180,E1 -435.98,E2 -435.98} C_VEL
LIN {X 0,Y 608.457,Z 315.143,A -85,B 0,C 180,E1 -438.676,E2 -438.676} C_VEL
LIN {X 0,Y 608.472,Z 322.485,A -85,B 0,C 180,E1 -439.75,E2 -439.75} C_VEL
LIN {X 0,Y 608.482,Z 400.434,A -85,B 0,C 180,E1 -440.694,E2 -440.694} C_VEL
LIN {X 0,Y 608.448,Z 410.068,A -85,B 0,C 180,E1 -440.903,E2 -440.903} C_VEL
LIN {X 0,Y 608.442,Z 421.613,A -85,B 0,C 180,E1 -441.28,E2 -441.28} C_VEL
LIN {X 0,Y 608.466,Z 432.23,A -85,B 0,C 180,E1 -441.782,E2 -441.782} C_VEL
LIN {X 0,Y 608.458,Z 440.54,A -85,B 0,C 180,E1 -442.283,E2 -442.283} C_VEL
LIN {X 0,Y 608.459,Z 448.399,A -85,B 0,C 180,E1 -442.867,E2 -442.867} C_VEL
LIN {X 0,Y 608.467,Z 455.358,A -85,B 0,C 180,E1 -443.496,E2 -443.496} C_VEL
LIN {X 0,Y 608.469,Z 463.19,A -85,B 0,C 180,E1 -444.366,E2 -444.366} C_VEL
LIN {X 0,Y 608.448,Z 469.026,A -85,B 0,C 180,E1 -445.196,E2 -445.196} C_VEL
LIN {X 0,Y 608.434,Z 473.63,A -85,B 0,C 180,E1 -446.026,E2 -446.026} C_VEL
LIN {X 0,Y 608.425,Z 476.621,A -85,B 0,C 180,E1 -446.689,E2 -446.689} C_VEL
LIN {X 0,Y 608.423,Z 478.931,A -85,B 0,C 180,E1 -447.352,E2 -447.352} C_VEL
LIN {X 0,Y 608.444,Z 480.678,A -85,B 0,C 180,E1 -448.014,E2 -448.014} C_VEL
LIN {X 0,Y 608.446,Z 481.933,A -85,B 0,C 180,E1 -448.676,E2 -448.676} C_VEL
LIN {X 0,Y 608.434,Z 482.714,A -85,B 0,C 180,E1 -449.338,E2 -449.338} C_VEL
LIN {X 0,Y 608.431,Z 483,A -85,B 0,C 180,E1 -450,E2 -450} C_VEL
LIN {X 0,Y 608.434,Z 482.714,A -85,B 0,C 180,E1 -450.662,E2 -450.662} C_VEL
LIN {X 0,Y 608.446,Z 481.934,A -85,B 0,C 180,E1 -451.324,E2 -451.324} C_VEL
LIN {X 0,Y 608.444,Z 480.678,A -85,B 0,C 180,E1 -451.986,E2 -451.986} C_VEL
LIN {X 0,Y 608.444,Z 477.786,A -85,B 0,C 180,E1 -452.979,E2 -452.979} C_VEL
LIN {X 0,Y 608.446,Z 475.147,A -85,B 0,C 180,E1 -453.642,E2 -453.642} C_VEL
LIN {X 0,Y 608.431,Z 469.985,A -85,B 0,C 180,E1 -454.638,E2 -454.638} C_VEL
LIN {X 0,Y 608.46,Z 464.43,A -85,B 0,C 180,E1 -455.468,E2 -455.468} C_VEL
LIN {X 0,Y 608.456,Z 456.674,A -85,B 0,C 180,E1 -456.375,E2 -456.375} C_VEL
LIN {X 0,Y 608.452,Z 449.416,A -85,B 0,C 180,E1 -457.049,E2 -457.049} C_VEL
LIN {X 0,Y 608.459,Z 441.761,A -85,B 0,C 180,E1 -457.633,E2 -457.633} C_VEL
LIN {X 0,Y 608.489,Z 433.721,A -85,B 0,C 180,E1 -458.134,E2 -458.134} C_VEL
LIN {X 0,Y 608.466,Z 425.391,A -85,B 0,C 180,E1 -458.552,E2 -458.552} C_VEL
LIN {X 0,Y 608.444,Z 416.891,A -85,B 0,C 180,E1 -458.887,E2 -458.887} C_VEL
LIN {X 0,Y 608.449,Z 407.588,A -85,B 0,C 180,E1 -459.159,E2 -459.159} C_VEL
LIN {X 0,Y 608.489,Z 396.553,A -85,B 0,C 180,E1 -459.368,E2 -459.368} C_VEL
LIN {X 0,Y 608.472,Z 322.487,A -85,B 0,C 180,E1 -460.25,E2 -460.25} C_VEL
LIN {X 0,Y 608.468,Z 302.476,A -85,B 0,C 180,E1 -463.186,E2 -463.186} C_VEL
LIN {X 0,Y 608.467,Z 284.048,A -85,B 0,C 180,E1 -465.921,E2 -465.921} C_VEL
LIN {X 0,Y 608.505,Z 265.412,A -85,B 0,C 180,E1 -468.725,E2 -468.725} C_VEL
LIN {X 0,Y 608.532,Z 247.193,A -85,B 0,C 180,E1 -471.511,E2 -471.511} C_VEL
LIN {X 0,Y 608.448,Z 244.502,A -85,B 0,C 180,E1 -471.96,E2 -471.96} C_VEL
LIN {X 0,Y 608.454,Z 244.501,A -85,B 0,C 180,E1 -474.571,E2 -474.571} C_VEL
LIN {X 0,Y 608.48,Z 244.507,A -85,B 0,C 180,E1 -477.207,E2 -477.207} C_VEL
LIN {X 0,Y 608.451,Z 244.501,A -85,B 0,C 180,E1 -479.968,E2 -479.968} C_VEL
LIN {X 0,Y 608.462,Z 244.501,A -85,B 0,C 180,E1 -482.879,E2 -482.879} C_VEL
LIN {X 0,Y 608.439,Z 244.511,A -85,B 0,C 180,E1 -485.278,E2 -485.278} C_VEL
LIN {X 0,Y 608.457,Z 244.504,A -85,B 0,C 180,E1 -487.747,E2 -487.747} C_VEL
LIN {X 0,Y 608.438,Z 244.501,A -85,B 0,C 180,E1 -490.327,E2 -490.327} C_VEL
LIN {X 0,Y 608.451,Z 244.502,A -85,B 0,C 180,E1 -492.96,E2 -492.96} C_VEL
LIN {X 0,Y 608.443,Z 244.507,A -85,B 0,C 180,E1 -495.737,E2 -495.737} C_VEL
LIN {X 0,Y 608.449,Z 244.504,A -85,B 0,C 180,E1 -497.937,E2 -497.937} C_VEL
LIN {X 0,Y 608.445,Z 244.5,A -85,B 0,C 180,E1 -500.705,E2 -500.705} C_VEL
LIN {X 0,Y 608.462,Z 244.501,A -85,B 0,C 180,E1 -503.084,E2 -503.084} C_VEL
LIN {X 0,Y 608.466,Z 244.507,A -85,B 0,C 180,E1 -505.529,E2 -505.529} C_VEL
LIN {X 0,Y 608.464,Z 244.505,A -85,B 0,C 180,E1 -507.904,E2 -507.904} C_VEL
LIN {X 0,Y 608.448,Z 244.502,A -85,B 0,C 180,E1 -510.218,E2 -510.218} C_VEL
LIN {X 0,Y 608.451,Z 244.499,A -85,B 0,C 180,E1 -512.798,E2 -512.798} C_VEL
LIN {X 0,Y 608.456,Z 244.504,A -85,B 0,C 180,E1 -515.428,E2 -515.428} C_VEL
LIN {X 0,Y 608.454,Z 244.502,A -85,B 0,C 180,E1 -518.306,E2 -518.306} C_VEL
LIN {X 0,Y 608.454,Z 244.5,A -85,B 0,C 180,E1 -521.129,E2 -521.129} C_VEL
LIN {X 0,Y 608.457,Z 244.51,A -85,B 0,C 180,E1 -523.904,E2 -523.904} C_VEL
LIN {X 0,Y 608.443,Z 244.501,A -85,B 0,C 180,E1 -526.641,E2 -526.641} C_VEL
LIN {X 0,Y 608.464,Z 244.499,A -85,B 0,C 180,E1 -529.348,E2 -529.348} C_VEL
LIN {X 0,Y 608.478,Z 244.507,A -85,B 0,C 180,E1 -532.031,E2 -532.031} C_VEL
LIN {X 0,Y 608.437,Z 244.502,A -85,B 0,C 180,E1 -534.696,E2 -534.696} C_VEL
LIN {X 0,Y 608.48,Z 244.497,A -85,B 0,C 180,E1 -537.35,E2 -537.35} C_VEL
LIN {X 0,Y 608.479,Z 244.505,A -85,B 0,C 180,E1 -539.998,E2 -539.998} C_VEL
LIN {X 0,Y 608.451,Z 244.502,A -85,B 0,C 180,E1 -542.646,E2 -542.646} C_VEL
LIN {X 0,Y 608.447,Z 244.5,A -85,B 0,C 180,E1 -545.3,E2 -545.3} C_VEL
LIN {X 0,Y 608.479,Z 244.503,A -85,B 0,C 180,E1 -547.964,E2 -547.964} C_VEL
LIN {X 0,Y 608.444,Z 244.501,A -85,B 0,C 180,E1 -549.438,E2 -549.438} C_VEL
LIN {X 0,Y 607.779,Z 244.591,A -85,B 0,C 180,E1 -549.991,E2 -549.991} C_VEL
LIN {X 0,Y 604.935,Z 244.948,A -85,B 0,C 180,E1 -550.888,E2 -550.888} C_VEL
LIN {X 0,Y 602.528,Z 245.248,A -85,B 0,C 180,E1 -551.609,E2 -551.609} C_VEL
LIN {X 0,Y 601.489,Z 245.376,A -85,B 0,C 180,E1 -552.166,E2 -552.166} C_VEL
LIN {X 0,Y 601.401,Z 245.383,A -85,B 0,C 180,E1 -552.354,E2 -552.354} C_VEL
LIN {X 0,Y 601.413,Z 245.378,A -85,B 0,C 180,E1 -554.895,E2 -554.895} C_VEL
LIN {X 0,Y 601.401,Z 245.379,A -85,B 0,C 180,E1 -556.984,E2 -556.984} C_VEL
LIN {X 0,Y 601.403,Z 245.378,A -85,B 0,C 180,E1 -559.096,E2 -559.096} C_VEL
LIN {X 0,Y 601.39,Z 245.379,A -85,B 0,C 180,E1 -561.237,E2 -561.237} C_VEL
LIN {X 0,Y 601.46,Z 245.376,A -85,B 0,C 180,E1 -564.137,E2 -564.137} C_VEL
LIN {X 0,Y 601.422,Z 245.376,A -85,B 0,C 180,E1 -567.109,E2 -567.109} C_VEL
LIN {X 0,Y 601.403,Z 245.377,A -85,B 0,C 180,E1 -569.39,E2 -569.39} C_VEL
LIN {X 0,Y 601.389,Z 245.38,A -85,B 0,C 180,E1 -571.724,E2 -571.724} C_VEL
LIN {X 0,Y 601.417,Z 245.379,A -85,B 0,C 180,E1 -574.115,E2 -574.115} C_VEL
LIN {X 0,Y 601.392,Z 245.39,A -85,B 0,C 180,E1 -576.579,E2 -576.579} C_VEL
LIN {X 0,Y 601.388,Z 245.382,A -85,B 0,C 180,E1 -579.124,E2 -579.124} C_VEL
LIN {X 0,Y 601.406,Z 245.377,A -85,B 0,C 180,E1 -581.762,E2 -581.762} C_VEL
LIN {X 0,Y 601.398,Z 245.386,A -85,B 0,C 180,E1 -584.533,E2 -584.533} C_VEL
LIN {X 0,Y 601.383,Z 245.382,A -85,B 0,C 180,E1 -587.327,E2 -587.327} C_VEL
LIN {X 0,Y 601.386,Z 245.38,A -85,B 0,C 180,E1 -590.003,E2 -590.003} C_VEL
LIN {X 0,Y 601.413,Z 245.384,A -85,B 0,C 180,E1 -592.614,E2 -592.614} C_VEL
LIN {X 0,Y 601.41,Z 245.384,A -85,B 0,C 180,E1 -595.068,E2 -595.068} C_VEL
LIN {X 0,Y 601.424,Z 245.548,A -85,B 0,C 180,E1 -596.385,E2 -596.385} C_VEL
LIN {X 0,Y 601.344,Z 257.86,A -85,B 0,C 180,E1 -599.054,E2 -599.054} C_VEL
LIN {X 0,Y 601.371,Z 270.438,A -85,B 0,C 180,E1 -601.751,E2 -601.751} C_VEL
LIN {X 0,Y 601.397,Z 274.873,A -85,B 0,C 180,E1 -602.696,E2 -602.696} C_VEL
LIN {X 0,Y 601.538,Z 288.081,A -85,B 0,C 180,E1 -602.87,E2 -602.87} C_VEL
LIN {X 0,Y 601.495,Z 349.649,A -85,B 0,C 180,E1 -603.617,E2 -603.617} C_VEL
LIN {X 0,Y 601.487,Z 358.953,A -85,B 0,C 180,E1 -603.814,E2 -603.814} C_VEL
LIN {X 0,Y 601.443,Z 368.712,A -85,B 0,C 180,E1 -604.118,E2 -604.118} C_VEL
LIN {X 0,Y 601.474,Z 379.268,A -85,B 0,C 180,E1 -604.57,E2 -604.57} C_VEL
LIN {X 0,Y 601.414,Z 390.06,A -85,B 0,C 180,E1 -605.204,E2 -605.204} C_VEL
LIN {X 0,Y 601.422,Z 396.869,A -85,B 0,C 180,E1 -605.701,E2 -605.701} C_VEL
LIN {X 0,Y 601.385,Z 404.771,A -85,B 0,C 180,E1 -606.406,E2 -606.406} C_VEL
LIN {X 0,Y 601.39,Z 411.431,A -85,B 0,C 180,E1 -607.135,E2 -607.135} C_VEL
LIN {X 0,Y 601.372,Z 418.115,A -85,B 0,C 180,E1 -608.039,E2 -608.039} C_VEL
LIN {X 0,Y 601.378,Z 423.616,A -85,B 0,C 180,E1 -609.021,E2 -609.021} C_VEL
LIN {X 0,Y 601.334,Z 427.109,A -85,B 0,C 180,E1 -609.832,E2 -609.832} C_VEL
LIN {X 0,Y 601.336,Z 429.491,A -85,B 0,C 180,E1 -610.544,E2 -610.544} C_VEL
LIN {X 0,Y 601.311,Z 431.793,A -85,B 0,C 180,E1 -611.605,E2 -611.605} C_VEL
LIN {X 0,Y 601.309,Z 432.682,A -85,B 0,C 180,E1 -612.309,E2 -612.309} C_VEL
LIN {X 0,Y 601.34,Z 432.998,A -85,B 0,C 180,E1 -613.012,E2 -613.012} C_VEL
LIN {X 0,Y 601.352,Z 432.715,A -85,B 0,C 180,E1 -613.711,E2 -613.711} C_VEL
LIN {X 0,Y 601.327,Z 431.903,A -85,B 0,C 180,E1 -614.407,E2 -614.407} C_VEL
LIN {X 0,Y 601.309,Z 430.57,A -85,B 0,C 180,E1 -615.1,E2 -615.1} C_VEL
LIN {X 0,Y 601.343,Z 427.311,A -85,B 0,C 180,E1 -616.199,E2 -616.199} C_VEL
LIN {X 0,Y 601.333,Z 423.154,A -85,B 0,C 180,E1 -617.17,E2 -617.17} C_VEL
LIN {X 0,Y 601.383,Z 417.08,A -85,B 0,C 180,E1 -618.199,E2 -618.199} C_VEL
LIN {X 0,Y 601.383,Z 411.167,A -85,B 0,C 180,E1 -618.987,E2 -618.987} C_VEL
LIN {X 0,Y 601.395,Z 405.979,A -85,B 0,C 180,E1 -619.564,E2 -619.564} C_VEL
LIN {X 0,Y 601.41,Z 398.608,A -85,B 0,C 180,E1 -620.245,E2 -620.245} C_VEL
LIN {X 0,Y 601.433,Z 390.739,A -85,B 0,C 180,E1 -620.839,E2 -620.839} C_VEL
LIN {X 0,Y 601.453,Z 380.948,A -85,B 0,C 180,E1 -621.432,E2 -621.432} C_VEL
LIN {X 0,Y 601.44,Z 369.653,A -85,B 0,C 180,E1 -621.939,E2 -621.939} C_VEL
LIN {X 0,Y 601.446,Z 359.768,A -85,B 0,C 180,E1 -622.256,E2 -622.256} C_VEL
LIN {X 0,Y 601.485,Z 349.954,A -85,B 0,C 180,E1 -622.468,E2 -622.468} C_VEL
LIN {X 0,Y 601.347,Z 275.045,A -85,B 0,C 180,E1 -623.378,E2 -623.378} C_VEL
LIN {X 0,Y 601.379,Z 262.771,A -85,B 0,C 180,E1 -625.979,E2 -625.979} C_VEL
LIN {X 0,Y 601.4,Z 250.345,A -85,B 0,C 180,E1 -628.661,E2 -628.661} C_VEL
LIN {X 0,Y 601.383,Z 245.383,A -85,B 0,C 180,E1 -629.749,E2 -629.749} C_VEL
LIN {X 0,Y 601.371,Z 245.382,A -85,B 0,C 180,E1 -632.009,E2 -632.009} C_VEL
LIN {X 0,Y 601.352,Z 245.385,A -85,B 0,C 180,E1 -634.021,E2 -634.021} C_VEL
LIN {X 0,Y 601.414,Z 245.378,A -85,B 0,C 180,E1 -636.676,E2 -636.676} C_VEL
LIN {X 0,Y 601.404,Z 245.387,A -85,B 0,C 180,E1 -639.416,E2 -639.416} C_VEL
LIN {X 0,Y 601.408,Z 245.386,A -85,B 0,C 180,E1 -641.459,E2 -641.459} C_VEL
LIN {X 0,Y 601.37,Z 245.382,A -85,B 0,C 180,E1 -644.207,E2 -644.207} C_VEL
LIN {X 0,Y 601.389,Z 245.383,A -85,B 0,C 180,E1 -646.987,E2 -646.987} C_VEL
LIN {X 0,Y 601.366,Z 245.386,A -85,B 0,C 180,E1 -649.811,E2 -649.811} C_VEL
LIN {X 0,Y 601.364,Z 245.383,A -85,B 0,C 180,E1 -652.685,E2 -652.685} C_VEL
LIN {X 0,Y 601.407,Z 245.385,A -85,B 0,C 180,E1 -655.619,E2 -655.619} C_VEL
LIN {X 0,Y 601.353,Z 245.388,A -85,B 0,C 180,E1 -657.871,E2 -657.871} C_VEL
LIN {X 0,Y 601.365,Z 245.383,A -85,B 0,C 180,E1 -660.168,E2 -660.168} C_VEL
LIN {X 0,Y 601.363,Z 245.383,A -85,B 0,C 180,E1 -662.714,E2 -662.714} C_VEL
LIN {X 0,Y 601.357,Z 245.387,A -85,B 0,C 180,E1 -665.113,E2 -665.113} C_VEL
LIN {X 0,Y 601.401,Z 245.386,A -85,B 0,C 180,E1 -667.422,E2 -667.422} C_VEL
LIN {X 0,Y 601.357,Z 245.387,A -85,B 0,C 180,E1 -670,E2 -670} C_VEL
LIN {X 0,Y 601.342,Z 245.385,A -85,B 0,C 180,E1 -672.589,E2 -672.589} C_VEL
LIN {X 0,Y 601.372,Z 245.381,A -85,B 0,C 180,E1 -674.535,E2 -674.535} C_VEL
LIN {X 0,Y 601.396,Z 245.385,A -85,B 0,C 180,E1 -677.411,E2 -677.411} C_VEL
LIN {X 0,Y 601.381,Z 245.385,A -85,B 0,C 180,E1 -680.007,E2 -680.007} C_VEL
LIN {X 0,Y 601.377,Z 245.381,A -85,B 0,C 180,E1 -682.626,E2 -682.626} C_VEL
LIN {X 0,Y 601.367,Z 245.384,A -85,B 0,C 180,E1 -685.069,E2 -685.069} C_VEL
LIN {X 0,Y 601.414,Z 245.383,A -85,B 0,C 180,E1 -687.487,E2 -687.487} C_VEL
LIN {X 0,Y 601.416,Z 245.385,A -85,B 0,C 180,E1 -689.854,E2 -689.854} C_VEL
LIN {X 0,Y 601.369,Z 245.382,A -85,B 0,C 180,E1 -692.647,E2 -692.647} C_VEL
LIN {X 0,Y 601.374,Z 245.383,A -85,B 0,C 180,E1 -695.124,E2 -695.124} C_VEL
LIN {X 0,Y 601.406,Z 245.381,A -85,B 0,C 180,E1 -697.398,E2 -697.398} C_VEL
LIN {X 0,Y 601.39,Z 245.384,A -85,B 0,C 180,E1 -700.193,E2 -700.193} C_VEL
LIN {X 0,Y 601.38,Z 245.384,A -85,B 0,C 180,E1 -702.314,E2 -702.314} C_VEL
LIN {X 0,Y 601.392,Z 245.574,A -85,B 0,C 180,E1 -703.39,E2 -703.39} C_VEL
LIN {X 0,Y 601.402,Z 258.54,A -85,B 0,C 180,E1 -706.202,E2 -706.202} C_VEL
LIN {X 0,Y 601.351,Z 271.729,A -85,B 0,C 180,E1 -709.026,E2 -709.026} C_VEL
LIN {X 0,Y 601.329,Z 274.866,A -85,B 0,C 180,E1 -709.693,E2 -709.693} C_VEL
LIN {X 0,Y 601.533,Z 282.46,A -85,B 0,C 180,E1 -709.803,E2 -709.803} C_VEL
LIN {X 0,Y 601.474,Z 350.488,A -85,B 0,C 180,E1 -710.63,E2 -710.63} C_VEL
LIN {X 0,Y 601.441,Z 361.775,A -85,B 0,C 180,E1 -710.884,E2 -710.884} C_VEL
LIN {X 0,Y 601.416,Z 372.622,A -85,B 0,C 180,E1 -711.265,E2 -711.265} C_VEL
LIN {X 0,Y 601.44,Z 382.998,A -85,B 0,C 180,E1 -711.773,E2 -711.773} C_VEL
LIN {X 0,Y 601.438,Z 392.386,A -85,B 0,C 180,E1 -712.364,E2 -712.364} C_VEL
LIN {X 0,Y 601.401,Z 401.878,A -85,B 0,C 180,E1 -713.123,E2 -713.123} C_VEL
LIN {X 0,Y 601.388,Z 410.005,A -85,B 0,C 180,E1 -713.965,E2 -713.965} C_VEL
LIN {X 0,Y 601.374,Z 415.309,A -85,B 0,C 180,E1 -714.638,E2 -714.638} C_VEL
LIN {X 0,Y 601.364,Z 419.741,A -85,B 0,C 180,E1 -715.31,E2 -715.31} C_VEL
LIN {X 0,Y 601.344,Z 423.441,A -85,B 0,C 180,E1 -715.981,E2 -715.981} C_VEL
LIN {X 0,Y 601.346,Z 427.645,A -85,B 0,C 180,E1 -716.988,E2 -716.988} C_VEL
LIN {X 0,Y 601.338,Z 430.584,A -85,B 0,C 180,E1 -717.993,E2 -717.993} C_VEL
LIN {X 0,Y 601.348,Z 431.882,A -85,B 0,C 180,E1 -718.663,E2 -718.663} C_VEL
LIN {X 0,Y 601.335,Z 432.703,A -85,B 0,C 180,E1 -719.333,E2 -719.333} C_VEL
LIN {X 0,Y 601.333,Z 432.988,A -85,B 0,C 180,E1 -720.002,E2 -720.002} C_VEL
LIN {X 0,Y 601.338,Z 432.743,A -85,B 0,C 180,E1 -720.672,E2 -720.672} C_VEL
LIN {X 0,Y 601.346,Z 432.003,A -85,B 0,C 180,E1 -721.341,E2 -721.341} C_VEL
LIN {X 0,Y 601.342,Z 430.788,A -85,B 0,C 180,E1 -722.011,E2 -722.011} C_VEL
LIN {X 0,Y 601.344,Z 427.939,A -85,B 0,C 180,E1 -723.017,E2 -723.017} C_VEL
LIN {X 0,Y 601.363,Z 425.344,A -85,B 0,C 180,E1 -723.687,E2 -723.687} C_VEL
LIN {X 0,Y 601.363,Z 420.23,A -85,B 0,C 180,E1 -724.694,E2 -724.694} C_VEL
LIN {X 0,Y 601.384,Z 414.731,A -85,B 0,C 180,E1 -725.535,E2 -725.535} C_VEL
LIN {X 0,Y 601.393,Z 407.619,A -85,B 0,C 180,E1 -726.4,E2 -726.4} C_VEL
LIN {X 0,Y 601.413,Z 398.936,A -85,B 0,C 180,E1 -727.219,E2 -727.219} C_VEL
LIN {X 0,Y 601.403,Z 391.185,A -85,B 0,C 180,E1 -727.81,E2 -727.81} C_VEL
LIN {X 0,Y 601.452,Z 381.531,A -85,B 0,C 180,E1 -728.401,E2 -728.401} C_VEL
LIN {X 0,Y 601.464,Z 370.539,A -85,B 0,C 180,E1 -728.908,E2 -728.908} C_VEL
LIN {X 0,Y 601.48,Z 359.326,A -85,B 0,C 180,E1 -729.268,E2 -729.268} C_VEL
LIN {X 0,Y 601.514,Z 349.238,A -85,B 0,C 180,E1 -729.48,E2 -729.48} C_VEL
LIN {X 0,Y 601.409,Z 275.354,A -85,B 0,C 180,E1 -730.374,E2 -730.374} C_VEL
LIN {X 0,Y 601.359,Z 274.669,A -85,B 0,C 180,E1 -730.438,E2 -730.438} C_VEL
LIN {X 0,Y 601.387,Z 261.862,A -85,B 0,C 180,E1 -733.174,E2 -733.174} C_VEL
LIN {X 0,Y 601.392,Z 249.055,A -85,B 0,C 180,E1 -735.941,E2 -735.941} C_VEL
LIN {X 0,Y 601.44,Z 245.376,A -85,B 0,C 180,E1 -736.756,E2 -736.756} C_VEL
LIN {X 0,Y 601.414,Z 245.377,A -85,B 0,C 180,E1 -739.101,E2 -739.101} C_VEL
LIN {X 0,Y 601.4,Z 245.378,A -85,B 0,C 180,E1 -741.241,E2 -741.241} C_VEL
LIN {X 0,Y 601.448,Z 245.38,A -85,B 0,C 180,E1 -744.142,E2 -744.142} C_VEL
LIN {X 0,Y 601.43,Z 245.375,A -85,B 0,C 180,E1 -747.113,E2 -747.113} C_VEL
LIN {X 0,Y 601.392,Z 245.379,A -85,B 0,C 180,E1 -749.396,E2 -749.396} C_VEL
LIN {X 0,Y 601.4,Z 245.379,A -85,B 0,C 180,E1 -751.728,E2 -751.728} C_VEL
LIN {X 0,Y 601.416,Z 245.381,A -85,B 0,C 180,E1 -754.12,E2 -754.12} C_VEL
LIN {X 0,Y 601.44,Z 245.373,A -85,B 0,C 180,E1 -757.382,E2 -757.382} C_VEL
LIN {X 0,Y 601.405,Z 245.38,A -85,B 0,C 180,E1 -759.997,E2 -759.997} C_VEL
LIN {X 0,Y 601.414,Z 245.385,A -85,B 0,C 180,E1 -762.671,E2 -762.671} C_VEL
LIN {X 0,Y 601.405,Z 245.377,A -85,B 0,C 180,E1 -765.48,E2 -765.48} C_VEL
LIN {X 0,Y 601.423,Z 245.383,A -85,B 0,C 180,E1 -768.408,E2 -768.408} C_VEL
LIN {X 0,Y 601.406,Z 245.384,A -85,B 0,C 180,E1 -770.873,E2 -770.873} C_VEL
LIN {X 0,Y 601.404,Z 245.378,A -85,B 0,C 180,E1 -773.417,E2 -773.417} C_VEL
LIN {X 0,Y 601.42,Z 245.377,A -85,B 0,C 180,E1 -776.067,E2 -776.067} C_VEL
LIN {X 0,Y 601.421,Z 245.383,A -85,B 0,C 180,E1 -778.546,E2 -778.546} C_VEL
LIN {X 0,Y 601.435,Z 245.375,A -85,B 0,C 180,E1 -781.373,E2 -781.373} C_VEL
LIN {X 0,Y 601.401,Z 245.378,A -85,B 0,C 180,E1 -783.636,E2 -783.636} C_VEL
LIN {X 0,Y 601.449,Z 245.372,A -85,B 0,C 180,E1 -785.859,E2 -785.859} C_VEL
LIN {X 0,Y 601.428,Z 245.472,A -85,B 0,C 180,E1 -787.952,E2 -787.952} C_VEL
LIN {X 0,Y 601.585,Z 257.557,A -85,B 0,C 180,E1 -789.84,E2 -789.84} C_VEL
LIN {X 0,Y 601.46,Z 275.985,A -85,B 0,C 180,E1 -792.664,E2 -792.664} C_VEL
LIN {X 0,Y 601.452,Z 292.109,A -85,B 0,C 180,E1 -795.104,E2 -795.104} C_VEL
LIN {X 0,Y 601.435,Z 310.536,A -85,B 0,C 180,E1 -797.858,E2 -797.858} C_VEL
LIN {X 0,Y 601.394,Z 322.603,A -85,B 0,C 180,E1 -799.638,E2 -799.638} C_VEL
LIN {X 0,Y 601.496,Z 399.133,A -85,B 0,C 180,E1 -800.564,E2 -800.564} C_VEL
LIN {X 0,Y 601.445,Z 408.408,A -85,B 0,C 180,E1 -800.754,E2 -800.754} C_VEL
LIN {X 0,Y 601.432,Z 416.885,A -85,B 0,C 180,E1 -801.008,E2 -801.008} C_VEL
LIN {X 0,Y 601.44,Z 425.389,A -85,B 0,C 180,E1 -801.347,E2 -801.347} C_VEL
LIN {X 0,Y 601.443,Z 433.719,A -85,B 0,C 180,E1 -801.77,E2 -801.77} C_VEL
LIN {X 0,Y 601.401,Z 441.759,A -85,B 0,C 180,E1 -802.277,E2 -802.277} C_VEL
LIN {X 0,Y 601.414,Z 449.413,A -85,B 0,C 180,E1 -802.868,E2 -802.868} C_VEL
LIN {X 0,Y 601.394,Z 457.158,A -85,B 0,C 180,E1 -803.598,E2 -803.598} C_VEL
LIN {X 0,Y 601.383,Z 464.43,A -85,B 0,C 180,E1 -804.467,E2 -804.467} C_VEL
LIN {X 0,Y 601.341,Z 469.985,A -85,B 0,C 180,E1 -805.307,E2 -805.307} C_VEL
LIN {X 0,Y 601.365,Z 475.146,A -85,B 0,C 180,E1 -806.315,E2 -806.315} C_VEL
LIN {X 0,Y 601.343,Z 477.786,A -85,B 0,C 180,E1 -806.985,E2 -806.985} C_VEL
LIN {X 0,Y 601.343,Z 480.679,A -85,B 0,C 180,E1 -807.991,E2 -807.991} C_VEL
LIN {X 0,Y 601.345,Z 481.934,A -85,B 0,C 180,E1 -808.66,E2 -808.66} C_VEL
LIN {X 0,Y 601.335,Z 482.713,A -85,B 0,C 180,E1 -809.33,E2 -809.33} C_VEL
LIN {X 0,Y 601.332,Z 483,A -85,B 0,C 180,E1 -810,E2 -810} C_VEL
LIN {X 0,Y 601.335,Z 482.713,A -85,B 0,C 180,E1 -810.67,E2 -810.67} C_VEL
LIN {X 0,Y 601.345,Z 481.935,A -85,B 0,C 180,E1 -811.339,E2 -811.339} C_VEL
LIN {X 0,Y 601.343,Z 480.679,A -85,B 0,C 180,E1 -812.009,E2 -812.009} C_VEL
LIN {X 0,Y 601.343,Z 477.787,A -85,B 0,C 180,E1 -813.015,E2 -813.015} C_VEL
LIN {X 0,Y 601.365,Z 475.147,A -85,B 0,C 180,E1 -813.685,E2 -813.685} C_VEL
LIN {X 0,Y 601.341,Z 469.986,A -85,B 0,C 180,E1 -814.693,E2 -814.693} C_VEL
LIN {X 0,Y 601.383,Z 464.431,A -85,B 0,C 180,E1 -815.533,E2 -815.533} C_VEL
LIN {X 0,Y 601.394,Z 457.158,A -85,B 0,C 180,E1 -816.402,E2 -816.402} C_VEL
LIN {X 0,Y 601.413,Z 449.418,A -85,B 0,C 180,E1 -817.132,E2 -817.132} C_VEL
LIN {X 0,Y 601.424,Z 441.764,A -85,B 0,C 180,E1 -817.723,E2 -817.723} C_VEL
LIN {X 0,Y 601.443,Z 433.724,A -85,B 0,C 180,E1 -818.23,E2 -818.23} C_VEL
LIN {X 0,Y 601.44,Z 425.395,A -85,B 0,C 180,E1 -818.653,E2 -818.653} C_VEL
LIN {X 0,Y 601.432,Z 416.893,A -85,B 0,C 180,E1 -818.992,E2 -818.992} C_VEL
LIN {X 0,Y 601.458,Z 406.759,A -85,B 0,C 180,E1 -819.288,E2 -819.288} C_VEL
LIN {X 0,Y 601.492,Z 395.068,A -85,B 0,C 180,E1 -819.499,E2 -819.499} C_VEL
LIN {X 0,Y 601.398,Z 322.487,A -85,B 0,C 180,E1 -820.372,E2 -820.372} C_VEL
LIN {X 0,Y 601.448,Z 303.628,A -85,B 0,C 180,E1 -823.171,E2 -823.171} C_VEL
LIN {X 0,Y 601.461,Z 285.2,A -85,B 0,C 180,E1 -825.938,E2 -825.938} C_VEL
LIN {X 0,Y 601.519,Z 266.089,A -85,B 0,C 180,E1 -828.847,E2 -828.847} C_VEL
LIN {X 0,Y 601.583,Z 249.497,A -85,B 0,C 180,E1 -831.412,E2 -831.412} C_VEL
LIN {X 0,Y 601.437,Z 245.377,A -85,B 0,C 180,E1 -832.092,E2 -832.092} C_VEL
LIN {X 0,Y 601.401,Z 245.383,A -85,B 0,C 180,E1 -834.879,E2 -834.879} C_VEL
LIN {X 0,Y 601.414,Z 245.386,A -85,B 0,C 180,E1 -837.361,E2 -837.361} C_VEL
LIN {X 0,Y 601.411,Z 245.386,A -85,B 0,C 180,E1 -839.393,E2 -839.393} C_VEL
LIN {X 0,Y 601.4,Z 245.382,A -85,B 0,C 180,E1 -841.727,E2 -841.727} C_VEL
LIN {X 0,Y 601.421,Z 245.376,A -85,B 0,C 180,E1 -844.119,E2 -844.119} C_VEL
LIN {X 0,Y 601.438,Z 245.384,A -85,B 0,C 180,E1 -847.382,E2 -847.382} C_VEL
LIN {X 0,Y 601.404,Z 245.38,A -85,B 0,C 180,E1 -849.996,E2 -849.996} C_VEL
LIN {X 0,Y 601.409,Z 245.377,A -85,B 0,C 180,E1 -852.67,E2 -852.67} C_VEL
LIN {X 0,Y 601.403,Z 245.388,A -85,B 0,C 180,E1 -855.479,E2 -855.479} C_VEL
LIN {X 0,Y 601.419,Z 245.376,A -85,B 0,C 180,E1 -858.407,E2 -858.407} C_VEL
LIN {X 0,Y 601.409,Z 245.378,A -85,B 0,C 180,E1 -860.872,E2 -860.872} C_VEL
LIN {X 0,Y 601.407,Z 245.385,A -85,B 0,C 180,E1 -863.416,E2 -863.416} C_VEL
LIN {X 0,Y 601.421,Z 245.379,A -85,B 0,C 180,E1 -866.066,E2 -866.066} C_VEL
LIN {X 0,Y 601.42,Z 245.375,A -85,B 0,C 180,E1 -868.545,E2 -868.545} C_VEL
LIN {X 0,Y 601.435,Z 245.379,A -85,B 0,C 180,E1 -871.372,E2 -871.372} C_VEL
LIN {X 0,Y 601.396,Z 245.383,A -85,B 0,C 180,E1 -874.136,E2 -874.136} C_VEL
LIN {X 0,Y 601.39,Z 245.379,A -85,B 0,C 180,E1 -876.587,E2 -876.587} C_VEL
LIN {X 0,Y 601.434,Z 245.378,A -85,B 0,C 180,E1 -879.477,E2 -879.477} C_VEL
LIN {X 0,Y 601.385,Z 245.383,A -85,B 0,C 180,E1 -882.31,E2 -882.31} C_VEL
LIN {X 0,Y 601.4,Z 245.38,A -85,B 0,C 180,E1 -884.407,E2 -884.407} C_VEL
LIN {X 0,Y 601.415,Z 245.376,A -85,B 0,C 180,E1 -887.17,E2 -887.17} C_VEL
LIN {X 0,Y 601.43,Z 245.384,A -85,B 0,C 180,E1 -889.903,E2 -889.903} C_VEL
LIN {X 0,Y 601.4,Z 245.379,A -85,B 0,C 180,E1 -892.612,E2 -892.612} C_VEL
LIN {X 0,Y 601.426,Z 245.375,A -85,B 0,C 180,E1 -895.306,E2 -895.306} C_VEL
LIN {X 0,Y 601.436,Z 245.383,A -85,B 0,C 180,E1 -897.989,E2 -897.989} C_VEL
LIN {X 0,Y 601.427,Z 245.376,A -85,B 0,C 180,E1 -900.667,E2 -900.667} C_VEL
LIN {X 0,Y 601.418,Z 245.376,A -85,B 0,C 180,E1 -903.347,E2 -903.347} C_VEL
LIN {X 0,Y 601.41,Z 245.385,A -85,B 0,C 180,E1 -906.035,E2 -906.035} C_VEL
LIN {X 0,Y 601.398,Z 245.381,A -85,B 0,C 180,E1 -908.736,E2 -908.736} C_VEL
LIN {X 0,Y 601.406,Z 245.377,A -85,B 0,C 180,E1 -911.456,E2 -911.456} C_VEL
LIN {X 0,Y 601.401,Z 245.383,A -85,B 0,C 180,E1 -912.354,E2 -912.354} C_VEL
LIN {X 0,Y 600.726,Z 245.464,A -85,B 0,C 180,E1 -912.914,E2 -912.914} C_VEL
LIN {X 0,Y 597.873,Z 245.821,A -85,B 0,C 180,E1 -913.821,E2 -913.821} C_VEL
LIN {X 0,Y 595.467,Z 246.123,A -85,B 0,C 180,E1 -914.552,E2 -914.552} C_VEL
LIN {X 0,Y 594.433,Z 246.246,A -85,B 0,C 180,E1 -915.115,E2 -915.115} C_VEL
LIN {X 0,Y 594.348,Z 246.256,A -85,B 0,C 180,E1 -915.306,E2 -915.306} C_VEL
LIN {X 0,Y 594.344,Z 246.26,A -85,B 0,C 180,E1 -917.902,E2 -917.902} C_VEL
LIN {X 0,Y 594.391,Z 246.255,A -85,B 0,C 180,E1 -920.773,E2 -920.773} C_VEL
LIN {X 0,Y 594.37,Z 246.254,A -85,B 0,C 180,E1 -923.702,E2 -923.702} C_VEL
LIN {X 0,Y 594.366,Z 246.261,A -85,B 0,C 180,E1 -926.697,E2 -926.697} C_VEL
LIN {X 0,Y 594.367,Z 246.257,A -85,B 0,C 180,E1 -928.996,E2 -928.996} C_VEL
LIN {X 0,Y 594.362,Z 246.255,A -85,B 0,C 180,E1 -931.64,E2 -931.64} C_VEL
LIN {X 0,Y 594.365,Z 246.265,A -85,B 0,C 180,E1 -934.577,E2 -934.577} C_VEL
LIN {X 0,Y 594.364,Z 246.257,A -85,B 0,C 180,E1 -937.084,E2 -937.084} C_VEL
LIN {X 0,Y 594.341,Z 246.257,A -85,B 0,C 180,E1 -939.77,E2 -939.77} C_VEL
LIN {X 0,Y 594.369,Z 246.26,A -85,B 0,C 180,E1 -942.371,E2 -942.371} C_VEL
LIN {X 0,Y 594.337,Z 246.261,A -85,B 0,C 180,E1 -945.189,E2 -945.189} C_VEL
LIN {X 0,Y 594.34,Z 246.258,A -85,B 0,C 180,E1 -947.622,E2 -947.622} C_VEL
LIN {X 0,Y 594.372,Z 246.257,A -85,B 0,C 180,E1 -950.319,E2 -950.319} C_VEL
LIN {X 0,Y 594.362,Z 246.264,A -85,B 0,C 180,E1 -952.912,E2 -952.912} C_VEL
LIN {X 0,Y 594.359,Z 246.256,A -85,B 0,C 180,E1 -955.858,E2 -955.858} C_VEL
LIN {X 0,Y 594.391,Z 246.268,A -85,B 0,C 180,E1 -956.341,E2 -956.341} C_VEL
LIN {X 0,Y 594.284,Z 258.578,A -85,B 0,C 180,E1 -959.041,E2 -959.041} C_VEL
LIN {X 0,Y 594.302,Z 269.484,A -85,B 0,C 180,E1 -961.409,E2 -961.409} C_VEL
LIN {X 0,Y 594.316,Z 274.933,A -85,B 0,C 180,E1 -962.584,E2 -962.584} C_VEL
LIN {X 0,Y 594.559,Z 291.202,A -85,B 0,C 180,E1 -962.787,E2 -962.787} C_VEL
LIN {X 0,Y 594.491,Z 350.006,A -85,B 0,C 180,E1 -963.511,E2 -963.511} C_VEL
LIN {X 0,Y 594.472,Z 359.405,A -85,B 0,C 180,E1 -963.715,E2 -963.715} C_VEL
LIN {X 0,Y 594.448,Z 370.054,A -85,B 0,C 180,E1 -964.059,E2 -964.059} C_VEL
LIN {X 0,Y 594.441,Z 380.426,A -85,B 0,C 180,E1 -964.529,E2 -964.529} C_VEL
LIN {X 0,Y 594.392,Z 389.741,A -85,B 0,C 180,E1 -965.088,E2 -965.088} C_VEL
LIN {X 0,Y 594.355,Z 397.086,A -85,B 0,C 180,E1 -965.631,E2 -965.631} C_VEL
LIN {X 0,Y 594.315,Z 404.436,A -85,B 0,C 180,E1 -966.293,E2 -966.293} C_VEL
LIN {X 0,Y 594.316,Z 411.155,A -85,B 0,C 180,E1 -967.031,E2 -967.031} C_VEL
LIN {X 0,Y 594.28,Z 417.887,A -85,B 0,C 180,E1 -967.946,E2 -967.946} C_VEL
LIN {X 0,Y 594.3,Z 422.964,A -85,B 0,C 180,E1 -968.832,E2 -968.832} C_VEL
LIN {X 0,Y 594.264,Z 426.327,A -85,B 0,C 180,E1 -969.581,E2 -969.581} C_VEL
LIN {X 0,Y 594.254,Z 429.852,A -85,B 0,C 180,E1 -970.662,E2 -970.662} C_VEL
LIN {X 0,Y 594.237,Z 431.489,A -85,B 0,C 180,E1 -971.378,E2 -971.378} C_VEL
LIN {X 0,Y 594.201,Z 432.49,A -85,B 0,C 180,E1 -972.09,E2 -972.09} C_VEL
LIN {X 0,Y 594.233,Z 432.899,A -85,B 0,C 180,E1 -973.318,E2 -973.318} C_VEL
LIN {X 0,Y 594.252,Z 432.191,A -85,B 0,C 180,E1 -974.216,E2 -974.216} C_VEL
LIN {X 0,Y 594.22,Z 431.057,A -85,B 0,C 180,E1 -974.918,E2 -974.918} C_VEL
LIN {X 0,Y 594.255,Z 428.581,A -85,B 0,C 180,E1 -975.861,E2 -975.861} C_VEL
LIN {X 0,Y 594.261,Z 425.628,A -85,B 0,C 180,E1 -976.667,E2 -976.667} C_VEL
LIN {X 0,Y 594.27,Z 422.414,A -85,B 0,C 180,E1 -977.362,E2 -977.362} C_VEL
LIN {X 0,Y 594.31,Z 417.294,A -85,B 0,C 180,E1 -978.23,E2 -978.23} C_VEL
LIN {X 0,Y 594.311,Z 412.118,A -85,B 0,C 180,E1 -978.944,E2 -978.944} C_VEL
LIN {X 0,Y 594.335,Z 406.287,A -85,B 0,C 180,E1 -979.611,E2 -979.611} C_VEL
LIN {X 0,Y 594.347,Z 398.979,A -85,B 0,C 180,E1 -980.299,E2 -980.299} C_VEL
LIN {X 0,Y 594.382,Z 391.184,A -85,B 0,C 180,E1 -980.901,E2 -980.901} C_VEL
LIN {X 0,Y 594.37,Z 383.007,A -85,B 0,C 180,E1 -981.415,E2 -981.415} C_VEL
LIN {X 0,Y 594.424,Z 372.602,A -85,B 0,C 180,E1 -981.929,E2 -981.929} C_VEL
LIN {X 0,Y 594.436,Z 360.951,A -85,B 0,C 180,E1 -982.335,E2 -982.335} C_VEL
LIN {X 0,Y 594.489,Z 350.491,A -85,B 0,C 180,E1 -982.571,E2 -982.571} C_VEL
LIN {X 0,Y 594.545,Z 294.867,A -85,B 0,C 180,E1 -983.26,E2 -983.26} C_VEL
LIN {X 0,Y 594.434,Z 276.148,A -85,B 0,C 180,E1 -983.487,E2 -983.487} C_VEL
LIN {X 0,Y 594.262,Z 274.869,A -85,B 0,C 180,E1 -983.521,E2 -983.521} C_VEL
LIN {X 0,Y 594.322,Z 263.71,A -85,B 0,C 180,E1 -985.931,E2 -985.931} C_VEL
LIN {X 0,Y 594.35,Z 251.281,A -85,B 0,C 180,E1 -988.645,E2 -988.645} C_VEL
LIN {X 0,Y 594.352,Z 246.258,A -85,B 0,C 180,E1 -989.788,E2 -989.788} C_VEL
LIN {X 0,Y 594.372,Z 246.256,A -85,B 0,C 180,E1 -992.711,E2 -992.711} C_VEL
LIN {X 0,Y 594.379,Z 246.261,A -85,B 0,C 180,E1 -995.428,E2 -995.428} C_VEL
LIN {X 0,Y 594.338,Z 246.258,A -85,B 0,C 180,E1 -998.158,E2 -998.158} C_VEL
LIN {X 0,Y 594.403,Z 246.256,A -85,B 0,C 180,E1 -1001.102,E2 -1001.102} C_VEL
LIN {X 0,Y 594.336,Z 246.258,A -85,B 0,C 180,E1 -1004.17,E2 -1004.17} C_VEL
LIN {X 0,Y 594.351,Z 246.264,A -85,B 0,C 180,E1 -1007.195,E2 -1007.195} C_VEL
LIN {X 0,Y 594.328,Z 246.26,A -85,B 0,C 180,E1 -1010.056,E2 -1010.056} C_VEL
LIN {X 0,Y 594.322,Z 246.263,A -85,B 0,C 180,E1 -1012.969,E2 -1012.969} C_VEL
LIN {X 0,Y 594.34,Z 246.264,A -85,B 0,C 180,E1 -1015.195,E2 -1015.195} C_VEL
LIN {X 0,Y 594.332,Z 246.269,A -85,B 0,C 180,E1 -1017.525,E2 -1017.525} C_VEL
LIN {X 0,Y 594.331,Z 246.259,A -85,B 0,C 180,E1 -1020.327,E2 -1020.327} C_VEL
LIN {X 0,Y 594.343,Z 246.259,A -85,B 0,C 180,E1 -1022.953,E2 -1022.953} C_VEL
LIN {X 0,Y 594.318,Z 246.269,A -85,B 0,C 180,E1 -1025.411,E2 -1025.411} C_VEL
LIN {X 0,Y 594.344,Z 246.261,A -85,B 0,C 180,E1 -1027.944,E2 -1027.944} C_VEL
LIN {X 0,Y 594.338,Z 246.258,A -85,B 0,C 180,E1 -1030.823,E2 -1030.823} C_VEL
LIN {X 0,Y 594.334,Z 246.265,A -85,B 0,C 180,E1 -1033.841,E2 -1033.841} C_VEL
LIN {X 0,Y 594.326,Z 246.259,A -85,B 0,C 180,E1 -1036.702,E2 -1036.702} C_VEL
LIN {X 0,Y 594.36,Z 246.262,A -85,B 0,C 180,E1 -1039.437,E2 -1039.437} C_VEL
LIN {X 0,Y 594.346,Z 246.258,A -85,B 0,C 180,E1 -1042.397,E2 -1042.397} C_VEL
LIN {X 0,Y 594.326,Z 246.259,A -85,B 0,C 180,E1 -1044.68,E2 -1044.68} C_VEL
LIN {X 0,Y 594.359,Z 246.257,A -85,B 0,C 180,E1 -1047.092,E2 -1047.092} C_VEL
LIN {X 0,Y 594.371,Z 246.264,A -85,B 0,C 180,E1 -1049.675,E2 -1049.675} C_VEL
LIN {X 0,Y 594.324,Z 246.26,A -85,B 0,C 180,E1 -1052.54,E2 -1052.54} C_VEL
LIN {X 0,Y 594.344,Z 246.257,A -85,B 0,C 180,E1 -1054.809,E2 -1054.809} C_VEL
LIN {X 0,Y 594.349,Z 246.259,A -85,B 0,C 180,E1 -1057.269,E2 -1057.269} C_VEL
LIN {X 0,Y 594.358,Z 246.264,A -85,B 0,C 180,E1 -1059.949,E2 -1059.949} C_VEL
LIN {X 0,Y 594.337,Z 246.264,A -85,B 0,C 180,E1 -1062.097,E2 -1062.097} C_VEL
LIN {X 0,Y 594.345,Z 246.293,A -85,B 0,C 180,E1 -1063.346,E2 -1063.346} C_VEL
LIN {X 0,Y 594.355,Z 259.866,A -85,B 0,C 180,E1 -1066.323,E2 -1066.323} C_VEL
LIN {X 0,Y 594.262,Z 272.668,A -85,B 0,C 180,E1 -1069.095,E2 -1069.095} C_VEL
LIN {X 0,Y 594.247,Z 274.869,A -85,B 0,C 180,E1 -1069.569,E2 -1069.569} C_VEL
LIN {X 0,Y 594.539,Z 280.717,A -85,B 0,C 180,E1 -1069.66,E2 -1069.66} C_VEL
LIN {X 0,Y 594.49,Z 350.549,A -85,B 0,C 180,E1 -1070.519,E2 -1070.519} C_VEL
LIN {X 0,Y 594.441,Z 361.806,A -85,B 0,C 180,E1 -1070.775,E2 -1070.775} C_VEL
LIN {X 0,Y 594.404,Z 372.637,A -85,B 0,C 180,E1 -1071.161,E2 -1071.161} C_VEL
LIN {X 0,Y 594.422,Z 383.025,A -85,B 0,C 180,E1 -1071.675,E2 -1071.675} C_VEL
LIN {X 0,Y 594.393,Z 392.408,A -85,B 0,C 180,E1 -1072.273,E2 -1072.273} C_VEL
LIN {X 0,Y 594.343,Z 401.871,A -85,B 0,C 180,E1 -1073.041,E2 -1073.041} C_VEL
LIN {X 0,Y 594.31,Z 408.745,A -85,B 0,C 180,E1 -1073.743,E2 -1073.743} C_VEL
LIN {X 0,Y 594.295,Z 415.313,A -85,B 0,C 180,E1 -1074.574,E2 -1074.574} C_VEL
LIN {X 0,Y 594.274,Z 419.743,A -85,B 0,C 180,E1 -1075.254,E2 -1075.254} C_VEL
LIN {X 0,Y 594.26,Z 423.446,A -85,B 0,C 180,E1 -1075.933,E2 -1075.933} C_VEL
LIN {X 0,Y 594.248,Z 427.652,A -85,B 0,C 180,E1 -1076.952,E2 -1076.952} C_VEL
LIN {X 0,Y 594.238,Z 430.591,A -85,B 0,C 180,E1 -1077.969,E2 -1077.969} C_VEL
LIN {X 0,Y 594.247,Z 431.89,A -85,B 0,C 180,E1 -1078.647,E2 -1078.647} C_VEL
LIN {X 0,Y 594.235,Z 432.707,A -85,B 0,C 180,E1 -1079.325,E2 -1079.325} C_VEL
LIN {X 0,Y 594.234,Z 432.977,A -85,B 0,C 180,E1 -1080.002,E2 -1080.002} C_VEL
LIN {X 0,Y 594.238,Z 432.751,A -85,B 0,C 180,E1 -1080.68,E2 -1080.68} C_VEL
LIN {X 0,Y 594.246,Z 432.009,A -85,B 0,C 180,E1 -1081.358,E2 -1081.358} C_VEL
LIN {X 0,Y 594.241,Z 430.794,A -85,B 0,C 180,E1 -1082.035,E2 -1082.035} C_VEL
LIN {X 0,Y 594.247,Z 427.942,A -85,B 0,C 180,E1 -1083.053,E2 -1083.053} C_VEL
LIN {X 0,Y 594.285,Z 425.344,A -85,B 0,C 180,E1 -1083.731,E2 -1083.731} C_VEL
LIN {X 0,Y 594.267,Z 420.227,A -85,B 0,C 180,E1 -1084.751,E2 -1084.751} C_VEL
LIN {X 0,Y 594.31,Z 414.724,A -85,B 0,C 180,E1 -1085.601,E2 -1085.601} C_VEL
LIN {X 0,Y 594.344,Z 407.613,A -85,B 0,C 180,E1 -1086.476,E2 -1086.476} C_VEL
LIN {X 0,Y 594.355,Z 398.941,A -85,B 0,C 180,E1 -1087.305,E2 -1087.305} C_VEL
LIN {X 0,Y 594.376,Z 389.975,A -85,B 0,C 180,E1 -1087.988,E2 -1087.988} C_VEL
LIN {X 0,Y 594.446,Z 379.906,A -85,B 0,C 180,E1 -1088.586,E2 -1088.586} C_VEL
LIN {X 0,Y 594.469,Z 369.372,A -85,B 0,C 180,E1 -1089.057,E2 -1089.057} C_VEL
LIN {X 0,Y 594.505,Z 358.506,A -85,B 0,C 180,E1 -1089.4,E2 -1089.4} C_VEL
LIN {X 0,Y 594.516,Z 347.929,A -85,B 0,C 180,E1 -1089.614,E2 -1089.614} C_VEL
LIN {X 0,Y 594.409,Z 275.979,A -85,B 0,C 180,E1 -1090.489,E2 -1090.489} C_VEL
LIN {X 0,Y 594.284,Z 274.866,A -85,B 0,C 180,E1 -1090.521,E2 -1090.521} C_VEL
LIN {X 0,Y 594.341,Z 261.86,A -85,B 0,C 180,E1 -1093.333,E2 -1093.333} C_VEL
LIN {X 0,Y 594.38,Z 249.052,A -85,B 0,C 180,E1 -1096.135,E2 -1096.135} C_VEL
LIN {X 0,Y 594.413,Z 246.251,A -85,B 0,C 180,E1 -1096.772,E2 -1096.772} C_VEL
LIN {X 0,Y 594.364,Z 246.255,A -85,B 0,C 180,E1 -1099.336,E2 -1099.336} C_VEL
LIN {X 0,Y 594.359,Z 246.256,A -85,B 0,C 180,E1 -1101.505,E2 -1101.505} C_VEL
LIN {X 0,Y 594.396,Z 246.26,A -85,B 0,C 180,E1 -1104.447,E2 -1104.447} C_VEL
LIN {X 0,Y 594.35,Z 246.257,A -85,B 0,C 180,E1 -1107.519,E2 -1107.519} C_VEL
LIN {X 0,Y 594.358,Z 246.257,A -85,B 0,C 180,E1 -1109.779,E2 -1109.779} C_VEL
LIN {X 0,Y 594.371,Z 246.26,A -85,B 0,C 180,E1 -1112.148,E2 -1112.148} C_VEL
LIN {X 0,Y 594.377,Z 246.261,A -85,B 0,C 180,E1 -1114.581,E2 -1114.581} C_VEL
LIN {X 0,Y 594.391,Z 246.251,A -85,B 0,C 180,E1 -1117.608,E2 -1117.608} C_VEL
LIN {X 0,Y 594.366,Z 246.264,A -85,B 0,C 180,E1 -1120.568,E2 -1120.568} C_VEL
LIN {X 0,Y 594.372,Z 246.254,A -85,B 0,C 180,E1 -1123.3,E2 -1123.3} C_VEL
LIN {X 0,Y 594.365,Z 246.258,A -85,B 0,C 180,E1 -1126.162,E2 -1126.162} C_VEL
LIN {X 0,Y 594.377,Z 246.255,A -85,B 0,C 180,E1 -1129.179,E2 -1129.179} C_VEL
LIN {X 0,Y 594.379,Z 246.255,A -85,B 0,C 180,E1 -1132.058,E2 -1132.058} C_VEL
LIN {X 0,Y 594.355,Z 246.267,A -85,B 0,C 180,E1 -1134.677,E2 -1134.677} C_VEL
LIN {X 0,Y 594.383,Z 246.256,A -85,B 0,C 180,E1 -1137.089,E2 -1137.089} C_VEL
LIN {X 0,Y 594.372,Z 246.254,A -85,B 0,C 180,E1 -1139.675,E2 -1139.675} C_VEL
LIN {X 0,Y 594.379,Z 246.26,A -85,B 0,C 180,E1 -1142.539,E2 -1142.539} C_VEL
LIN {X 0,Y 594.392,Z 246.252,A -85,B 0,C 180,E1 -1145.554,E2 -1145.554} C_VEL
LIN {X 0,Y 594.396,Z 246.328,A -85,B 0,C 180,E1 -1147.813,E2 -1147.813} C_VEL
LIN {X 0,Y 594.637,Z 252.62,A -85,B 0,C 180,E1 -1148.818,E2 -1148.818} C_VEL
LIN {X 0,Y 594.567,Z 270.226,A -85,B 0,C 180,E1 -1151.567,E2 -1151.567} C_VEL
LIN {X 0,Y 594.417,Z 288.653,A -85,B 0,C 180,E1 -1154.396,E2 -1154.396} C_VEL
LIN {X 0,Y 594.389,Z 305.929,A -85,B 0,C 180,E1 -1157.017,E2 -1157.017} C_VEL
LIN {X 0,Y 594.344,Z 322.603,A -85,B 0,C 180,E1 -1159.514,E2 -1159.514} C_VEL
LIN {X 0,Y 594.592,Z 343.173,A -85,B 0,C 180,E1 -1159.766,E2 -1159.766} C_VEL
LIN {X 0,Y 594.48,Z 400.431,A -85,B 0,C 180,E1 -1160.473,E2 -1160.473} C_VEL
LIN {X 0,Y 594.443,Z 410.898,A -85,B 0,C 180,E1 -1160.708,E2 -1160.708} C_VEL
LIN {X 0,Y 594.413,Z 423.53,A -85,B 0,C 180,E1 -1161.158,E2 -1161.158} C_VEL
LIN {X 0,Y 594.407,Z 432.234,A -85,B 0,C 180,E1 -1161.586,E2 -1161.586} C_VEL
LIN {X 0,Y 594.375,Z 440.544,A -85,B 0,C 180,E1 -1162.099,E2 -1162.099} C_VEL
LIN {X 0,Y 594.351,Z 448.4,A -85,B 0,C 180,E1 -1162.697,E2 -1162.697} C_VEL
LIN {X 0,Y 594.343,Z 455.516,A -85,B 0,C 180,E1 -1163.357,E2 -1163.357} C_VEL
LIN {X 0,Y 594.318,Z 463.189,A -85,B 0,C 180,E1 -1164.231,E2 -1164.231} C_VEL
LIN {X 0,Y 594.256,Z 469.985,A -85,B 0,C 180,E1 -1165.251,E2 -1165.251} C_VEL
LIN {X 0,Y 594.287,Z 475.146,A -85,B 0,C 180,E1 -1166.271,E2 -1166.271} C_VEL
LIN {X 0,Y 594.246,Z 477.787,A -85,B 0,C 180,E1 -1166.949,E2 -1166.949} C_VEL
LIN {X 0,Y 594.242,Z 480.679,A -85,B 0,C 180,E1 -1167.967,E2 -1167.967} C_VEL
LIN {X 0,Y 594.245,Z 481.935,A -85,B 0,C 180,E1 -1168.644,E2 -1168.644} C_VEL
LIN {X 0,Y 594.235,Z 482.712,A -85,B 0,C 180,E1 -1169.322,E2 -1169.322} C_VEL
LIN {X 0,Y 594.233,Z 483,A -85,B 0,C 180,E1 -1170,E2 -1170} C_VEL
LIN {X 0,Y 594.235,Z 482.712,A -85,B 0,C 180,E1 -1170.678,E2 -1170.678} C_VEL
LIN {X 0,Y 594.245,Z 481.935,A -85,B 0,C 180,E1 -1171.355,E2 -1171.355} C_VEL
LIN {X 0,Y 594.242,Z 480.68,A -85,B 0,C 180,E1 -1172.033,E2 -1172.033} C_VEL
LIN {X 0,Y 594.246,Z 477.787,A -85,B 0,C 180,E1 -1173.051,E2 -1173.051} C_VEL
LIN {X 0,Y 594.287,Z 475.147,A -85,B 0,C 180,E1 -1173.729,E2 -1173.729} C_VEL
LIN {X 0,Y 594.256,Z 469.986,A -85,B 0,C 180,E1 -1174.749,E2 -1174.749} C_VEL
LIN {X 0,Y 594.309,Z 464.431,A -85,B 0,C 180,E1 -1175.599,E2 -1175.599} C_VEL
LIN {X 0,Y 594.345,Z 457.158,A -85,B 0,C 180,E1 -1176.479,E2 -1176.479} C_VEL
LIN {X 0,Y 594.354,Z 449.419,A -85,B 0,C 180,E1 -1177.217,E2 -1177.217} C_VEL
LIN {X 0,Y 594.359,Z 441.767,A -85,B 0,C 180,E1 -1177.815,E2 -1177.815} C_VEL
LIN {X 0,Y 594.419,Z 433.727,A -85,B 0,C 180,E1 -1178.328,E2 -1178.328} C_VEL
LIN {X 0,Y 594.423,Z 425.398,A -85,B 0,C 180,E1 -1178.756,E2 -1178.756} C_VEL
LIN {X 0,Y 594.421,Z 416.895,A -85,B 0,C 180,E1 -1179.099,E2 -1179.099} C_VEL
LIN {X 0,Y 594.468,Z 406.758,A -85,B 0,C 180,E1 -1179.398,E2 -1179.398} C_VEL
LIN {X 0,Y 594.51,Z 395.068,A -85,B 0,C 180,E1 -1179.612,E2 -1179.612} C_VEL
LIN {X 0,Y 594.448,Z 323.52,A -85,B 0,C 180,E1 -1180.473,E2 -1180.473} C_VEL
LIN {X 0,Y 594.346,Z 322.487,A -85,B 0,C 180,E1 -1180.496,E2 -1180.496} C_VEL
LIN {X 0,Y 594.409,Z 303.628,A -85,B 0,C 180,E1 -1183.33,E2 -1183.33} C_VEL
LIN {X 0,Y 594.495,Z 284.048,A -85,B 0,C 180,E1 -1186.306,E2 -1186.306} C_VEL
LIN {X 0,Y 594.542,Z 265.965,A -85,B 0,C 180,E1 -1189.096,E2 -1189.096} C_VEL
LIN {X 0,Y 594.645,Z 249.497,A -85,B 0,C 180,E1 -1191.675,E2 -1191.675} C_VEL
LIN {X 0,Y 594.382,Z 246.258,A -85,B 0,C 180,E1 -1192.233,E2 -1192.233} C_VEL
LIN {X 0,Y 594.371,Z 246.265,A -85,B 0,C 180,E1 -1195.193,E2 -1195.193} C_VEL
LIN {X 0,Y 594.371,Z 246.26,A -85,B 0,C 180,E1 -1197.523,E2 -1197.523} C_VEL
LIN {X 0,Y 594.373,Z 246.253,A -85,B 0,C 180,E1 -1200.325,E2 -1200.325} C_VEL
LIN {X 0,Y 594.381,Z 246.256,A -85,B 0,C 180,E1 -1202.95,E2 -1202.95} C_VEL
LIN {X 0,Y 594.352,Z 246.266,A -85,B 0,C 180,E1 -1205.409,E2 -1205.409} C_VEL
LIN {X 0,Y 594.379,Z 246.255,A -85,B 0,C 180,E1 -1207.941,E2 -1207.941} C_VEL
LIN {X 0,Y 594.376,Z 246.255,A -85,B 0,C 180,E1 -1210.821,E2 -1210.821} C_VEL
LIN {X 0,Y 594.369,Z 246.262,A -85,B 0,C 180,E1 -1213.299,E2 -1213.299} C_VEL
LIN {X 0,Y 594.364,Z 246.256,A -85,B 0,C 180,E1 -1216.161,E2 -1216.161} C_VEL
LIN {X 0,Y 594.378,Z 246.253,A -85,B 0,C 180,E1 -1218.535,E2 -1218.535} C_VEL
LIN {X 0,Y 594.376,Z 246.259,A -85,B 0,C 180,E1 -1221.297,E2 -1221.297} C_VEL
LIN {X 0,Y 594.353,Z 246.264,A -85,B 0,C 180,E1 -1223.754,E2 -1223.754} C_VEL
LIN {X 0,Y 594.368,Z 246.256,A -85,B 0,C 180,E1 -1226.237,E2 -1226.237} C_VEL
LIN {X 0,Y 594.37,Z 246.253,A -85,B 0,C 180,E1 -1228.649,E2 -1228.649} C_VEL
LIN {X 0,Y 594.384,Z 246.253,A -85,B 0,C 180,E1 -1231.042,E2 -1231.042} C_VEL
LIN {X 0,Y 594.361,Z 246.26,A -85,B 0,C 180,E1 -1234.054,E2 -1234.054} C_VEL
LIN {X 0,Y 594.373,Z 246.256,A -85,B 0,C 180,E1 -1236.294,E2 -1236.294} C_VEL
LIN {X 0,Y 594.408,Z 246.25,A -85,B 0,C 180,E1 -1239.223,E2 -1239.223} C_VEL
LIN {X 0,Y 594.343,Z 246.263,A -85,B 0,C 180,E1 -1242.093,E2 -1242.093} C_VEL
LIN {X 0,Y 594.358,Z 246.26,A -85,B 0,C 180,E1 -1244.217,E2 -1244.217} C_VEL
LIN {X 0,Y 594.372,Z 246.257,A -85,B 0,C 180,E1 -1246.319,E2 -1246.319} C_VEL
LIN {X 0,Y 594.377,Z 246.252,A -85,B 0,C 180,E1 -1249.093,E2 -1249.093} C_VEL
LIN {X 0,Y 594.415,Z 246.256,A -85,B 0,C 180,E1 -1251.841,E2 -1251.841} C_VEL
LIN {X 0,Y 594.373,Z 246.255,A -85,B 0,C 180,E1 -1254.57,E2 -1254.57} C_VEL
LIN {X 0,Y 594.405,Z 246.249,A -85,B 0,C 180,E1 -1257.287,E2 -1257.287} C_VEL
LIN {X 0,Y 594.416,Z 246.257,A -85,B 0,C 180,E1 -1259.998,E2 -1259.998} C_VEL
LIN {X 0,Y 594.387,Z 246.253,A -85,B 0,C 180,E1 -1262.709,E2 -1262.709} C_VEL
LIN {X 0,Y 594.379,Z 246.252,A -85,B 0,C 180,E1 -1265.425,E2 -1265.425} C_VEL
LIN {X 0,Y 594.41,Z 246.259,A -85,B 0,C 180,E1 -1268.154,E2 -1268.154} C_VEL
LIN {X 0,Y 594.375,Z 246.253,A -85,B 0,C 180,E1 -1271.066,E2 -1271.066} C_VEL
LIN {X 0,Y 594.37,Z 246.255,A -85,B 0,C 180,E1 -1273.676,E2 -1273.676} C_VEL
LIN {X 0,Y 594.348,Z 246.256,A -85,B 0,C 180,E1 -1275.306,E2 -1275.306} C_VEL
LIN {X 0,Y 593.677,Z 246.344,A -85,B 0,C 180,E1 -1275.872,E2 -1275.872} C_VEL
LIN {X 0,Y 590.814,Z 246.704,A -85,B 0,C 180,E1 -1276.79,E2 -1276.79} C_VEL
LIN {X 0,Y 588.404,Z 247.006,A -85,B 0,C 180,E1 -1277.528,E2 -1277.528} C_VEL
LIN {X 0,Y 587.378,Z 247.131,A -85,B 0,C 180,E1 -1278.098,E2 -1278.098} C_VEL
LIN {X 0,Y 587.3,Z 247.139,A -85,B 0,C 180,E1 -1278.291,E2 -1278.291} C_VEL
LIN {X 0,Y 587.321,Z 247.133,A -85,B 0,C 180,E1 -1281.035,E2 -1281.035} C_VEL
LIN {X 0,Y 587.305,Z 247.134,A -85,B 0,C 180,E1 -1283.256,E2 -1283.256} C_VEL
LIN {X 0,Y 587.317,Z 247.132,A -85,B 0,C 180,E1 -1285.514,E2 -1285.514} C_VEL
LIN {X 0,Y 587.337,Z 247.131,A -85,B 0,C 180,E1 -1287.815,E2 -1287.815} C_VEL
LIN {X 0,Y 587.329,Z 247.142,A -85,B 0,C 180,E1 -1290.508,E2 -1290.508} C_VEL
LIN {X 0,Y 587.317,Z 247.133,A -85,B 0,C 180,E1 -1293.394,E2 -1293.394} C_VEL
LIN {X 0,Y 587.3,Z 247.135,A -85,B 0,C 180,E1 -1295.895,E2 -1295.895} C_VEL
LIN {X 0,Y 587.313,Z 247.141,A -85,B 0,C 180,E1 -1298.476,E2 -1298.476} C_VEL
LIN {X 0,Y 587.314,Z 247.135,A -85,B 0,C 180,E1 -1301.154,E2 -1301.154} C_VEL
LIN {X 0,Y 587.297,Z 247.135,A -85,B 0,C 180,E1 -1303.948,E2 -1303.948} C_VEL
LIN {X 0,Y 587.298,Z 247.143,A -85,B 0,C 180,E1 -1306.878,E2 -1306.878} C_VEL
LIN {X 0,Y 587.292,Z 247.136,A -85,B 0,C 180,E1 -1309.744,E2 -1309.744} C_VEL
LIN {X 0,Y 587.32,Z 247.137,A -85,B 0,C 180,E1 -1312.391,E2 -1312.391} C_VEL
LIN {X 0,Y 587.323,Z 247.141,A -85,B 0,C 180,E1 -1314.944,E2 -1314.944} C_VEL
LIN {X 0,Y 587.369,Z 247.219,A -85,B 0,C 180,E1 -1316.349,E2 -1316.349} C_VEL
LIN {X 0,Y 587.223,Z 259.295,A -85,B 0,C 180,E1 -1319.027,E2 -1319.027} C_VEL
LIN {X 0,Y 587.227,Z 270.085,A -85,B 0,C 180,E1 -1321.398,E2 -1321.398} C_VEL
LIN {X 0,Y 587.238,Z 274.882,A -85,B 0,C 180,E1 -1322.445,E2 -1322.445} C_VEL
LIN {X 0,Y 587.573,Z 280.461,A -85,B 0,C 180,E1 -1322.533,E2 -1322.533} C_VEL
LIN {X 0,Y 587.504,Z 349.879,A -85,B 0,C 180,E1 -1323.395,E2 -1323.395} C_VEL
LIN {X 0,Y 587.482,Z 359.621,A -85,B 0,C 180,E1 -1323.609,E2 -1323.609} C_VEL
LIN {X 0,Y 587.443,Z 370.441,A -85,B 0,C 180,E1 -1323.965,E2 -1323.965} C_VEL
LIN {X 0,Y 587.411,Z 381.481,A -85,B 0,C 180,E1 -1324.487,E2 -1324.487} C_VEL
LIN {X 0,Y 587.329,Z 390.587,A -85,B 0,C 180,E1 -1325.052,E2 -1325.052} C_VEL
LIN {X 0,Y 587.286,Z 398.425,A -85,B 0,C 180,E1 -1325.655,E2 -1325.655} C_VEL
LIN {X 0,Y 587.251,Z 405.945,A -85,B 0,C 180,E1 -1326.365,E2 -1326.365} C_VEL
LIN {X 0,Y 587.241,Z 413.953,A -85,B 0,C 180,E1 -1327.309,E2 -1327.309} C_VEL
LIN {X 0,Y 587.187,Z 419.883,A -85,B 0,C 180,E1 -1328.221,E2 -1328.221} C_VEL
LIN {X 0,Y 587.204,Z 423.88,A -85,B 0,C 180,E1 -1328.983,E2 -1328.983} C_VEL
LIN {X 0,Y 587.178,Z 426.891,A -85,B 0,C 180,E1 -1329.69,E2 -1329.69} C_VEL
LIN {X 0,Y 587.155,Z 429.309,A -85,B 0,C 180,E1 -1330.419,E2 -1330.419} C_VEL
LIN {X 0,Y 587.141,Z 431.047,A -85,B 0,C 180,E1 -1331.144,E2 -1331.144} C_VEL
LIN {X 0,Y 587.117,Z 432.201,A -85,B 0,C 180,E1 -1331.867,E2 -1331.867} C_VEL
LIN {X 0,Y 587.12,Z 432.817,A -85,B 0,C 180,E1 -1332.587,E2 -1332.587} C_VEL
LIN {X 0,Y 587.133,Z 432.907,A -85,B 0,C 180,E1 -1333.305,E2 -1333.305} C_VEL
LIN {X 0,Y 587.155,Z 432.479,A -85,B 0,C 180,E1 -1334.02,E2 -1334.02} C_VEL
LIN {X 0,Y 587.134,Z 431.489,A -85,B 0,C 180,E1 -1334.732,E2 -1334.732} C_VEL
LIN {X 0,Y 587.177,Z 428.913,A -85,B 0,C 180,E1 -1335.795,E2 -1335.795} C_VEL
LIN {X 0,Y 587.174,Z 426.519,A -85,B 0,C 180,E1 -1336.503,E2 -1336.503} C_VEL
LIN {X 0,Y 587.187,Z 421.613,A -85,B 0,C 180,E1 -1337.559,E2 -1337.559} C_VEL
LIN {X 0,Y 587.21,Z 416.318,A -85,B 0,C 180,E1 -1338.436,E2 -1338.436} C_VEL
LIN {X 0,Y 587.235,Z 411.128,A -85,B 0,C 180,E1 -1339.135,E2 -1339.135} C_VEL
LIN {X 0,Y 587.272,Z 404.881,A -85,B 0,C 180,E1 -1339.833,E2 -1339.833} C_VEL
LIN {X 0,Y 587.282,Z 397.309,A -85,B 0,C 180,E1 -1340.529,E2 -1340.529} C_VEL
LIN {X 0,Y 587.385,Z 387.902,A -85,B 0,C 180,E1 -1341.225,E2 -1341.225} C_VEL
LIN {X 0,Y 587.373,Z 378.859,A -85,B 0,C 180,E1 -1341.745,E2 -1341.745} C_VEL
LIN {X 0,Y 587.395,Z 368.985,A -85,B 0,C 180,E1 -1342.178,E2 -1342.178} C_VEL
LIN {X 0,Y 587.433,Z 359.484,A -85,B 0,C 180,E1 -1342.485,E2 -1342.485} C_VEL
LIN {X 0,Y 587.497,Z 351.028,A -85,B 0,C 180,E1 -1342.676,E2 -1342.676} C_VEL
LIN {X 0,Y 587.561,Z 318.447,A -85,B 0,C 180,E1 -1343.095,E2 -1343.095} C_VEL
LIN {X 0,Y 587.416,Z 276.43,A -85,B 0,C 180,E1 -1343.609,E2 -1343.609} C_VEL
LIN {X 0,Y 587.21,Z 274.864,A -85,B 0,C 180,E1 -1343.649,E2 -1343.649} C_VEL
LIN {X 0,Y 587.279,Z 263.085,A -85,B 0,C 180,E1 -1346.226,E2 -1346.226} C_VEL
LIN {X 0,Y 587.302,Z 252.218,A -85,B 0,C 180,E1 -1348.629,E2 -1348.629} C_VEL
LIN {X 0,Y 587.324,Z 247.134,A -85,B 0,C 180,E1 -1349.786,E2 -1349.786} C_VEL
LIN {X 0,Y 587.339,Z 247.132,A -85,B 0,C 180,E1 -1352.744,E2 -1352.744} C_VEL
LIN {X 0,Y 587.339,Z 247.137,A -85,B 0,C 180,E1 -1355.493,E2 -1355.493} C_VEL
LIN {X 0,Y 587.3,Z 247.134,A -85,B 0,C 180,E1 -1358.256,E2 -1358.256} C_VEL
LIN {X 0,Y 587.351,Z 247.136,A -85,B 0,C 180,E1 -1361.156,E2 -1361.156} C_VEL
LIN {X 0,Y 587.293,Z 247.135,A -85,B 0,C 180,E1 -1364.249,E2 -1364.249} C_VEL
LIN {X 0,Y 587.317,Z 247.143,A -85,B 0,C 180,E1 -1367.407,E2 -1367.407} C_VEL
LIN {X 0,Y 587.28,Z 247.137,A -85,B 0,C 180,E1 -1370.307,E2 -1370.307} C_VEL
LIN {X 0,Y 587.276,Z 247.145,A -85,B 0,C 180,E1 -1373.261,E2 -1373.261} C_VEL
LIN {X 0,Y 587.297,Z 247.145,A -85,B 0,C 180,E1 -1375.519,E2 -1375.519} C_VEL
LIN {X 0,Y 587.299,Z 247.139,A -85,B 0,C 180,E1 -1377.82,E2 -1377.82} C_VEL
LIN {X 0,Y 587.286,Z 247.136,A -85,B 0,C 180,E1 -1380.509,E2 -1380.509} C_VEL
LIN {X 0,Y 587.306,Z 247.142,A -85,B 0,C 180,E1 -1383.399,E2 -1383.399} C_VEL
LIN {X 0,Y 587.256,Z 247.144,A -85,B 0,C 180,E1 -1385.903,E2 -1385.903} C_VEL
LIN {X 0,Y 587.284,Z 247.136,A -85,B 0,C 180,E1 -1388.483,E2 -1388.483} C_VEL
LIN {X 0,Y 587.305,Z 247.138,A -85,B 0,C 180,E1 -1391.16,E2 -1391.16} C_VEL
LIN {X 0,Y 587.286,Z 247.139,A -85,B 0,C 180,E1 -1394.115,E2 -1394.115} C_VEL
LIN {X 0,Y 587.282,Z 247.138,A -85,B 0,C 180,E1 -1396.996,E2 -1396.996} C_VEL
LIN {X 0,Y 587.295,Z 247.144,A -85,B 0,C 180,E1 -1399.749,E2 -1399.749} C_VEL
LIN {X 0,Y 587.301,Z 247.135,A -85,B 0,C 180,E1 -1402.393,E2 -1402.393} C_VEL
LIN {X 0,Y 587.298,Z 247.135,A -85,B 0,C 180,E1 -1404.947,E2 -1404.947} C_VEL
LIN {X 0,Y 587.32,Z 247.138,A -85,B 0,C 180,E1 -1407.424,E2 -1407.424} C_VEL
LIN {X 0,Y 587.316,Z 247.142,A -85,B 0,C 180,E1 -1409.833,E2 -1409.833} C_VEL
LIN {X 0,Y 587.287,Z 247.138,A -85,B 0,C 180,E1 -1412.32,E2 -1412.32} C_VEL
LIN {X 0,Y 587.342,Z 247.134,A -85,B 0,C 180,E1 -1415.423,E2 -1415.423} C_VEL
LIN {X 0,Y 587.305,Z 247.138,A -85,B 0,C 180,E1 -1418.228,E2 -1418.228} C_VEL
LIN {X 0,Y 587.324,Z 247.133,A -85,B 0,C 180,E1 -1421.153,E2 -1421.153} C_VEL
LIN {X 0,Y 587.316,Z 247.267,A -85,B 0,C 180,E1 -1423.358,E2 -1423.358} C_VEL
LIN {X 0,Y 587.301,Z 261.469,A -85,B 0,C 180,E1 -1426.508,E2 -1426.508} C_VEL
LIN {X 0,Y 587.185,Z 274.713,A -85,B 0,C 180,E1 -1429.408,E2 -1429.408} C_VEL
LIN {X 0,Y 587.197,Z 275.099,A -85,B 0,C 180,E1 -1429.46,E2 -1429.46} C_VEL
LIN {X 0,Y 587.566,Z 281.137,A -85,B 0,C 180,E1 -1429.541,E2 -1429.541} C_VEL
LIN {X 0,Y 587.5,Z 350.609,A -85,B 0,C 180,E1 -1430.405,E2 -1430.405} C_VEL
LIN {X 0,Y 587.451,Z 361.827,A -85,B 0,C 180,E1 -1430.665,E2 -1430.665} C_VEL
LIN {X 0,Y 587.402,Z 372.645,A -85,B 0,C 180,E1 -1431.055,E2 -1431.055} C_VEL
LIN {X 0,Y 587.39,Z 383.052,A -85,B 0,C 180,E1 -1431.574,E2 -1431.574} C_VEL
LIN {X 0,Y 587.354,Z 392.431,A -85,B 0,C 180,E1 -1432.18,E2 -1432.18} C_VEL
LIN {X 0,Y 587.297,Z 401.863,A -85,B 0,C 180,E1 -1432.957,E2 -1432.957} C_VEL
LIN {X 0,Y 587.267,Z 410.022,A -85,B 0,C 180,E1 -1433.819,E2 -1433.819} C_VEL
LIN {X 0,Y 587.221,Z 415.316,A -85,B 0,C 180,E1 -1434.508,E2 -1434.508} C_VEL
LIN {X 0,Y 587.187,Z 419.746,A -85,B 0,C 180,E1 -1435.196,E2 -1435.196} C_VEL
LIN {X 0,Y 587.181,Z 423.451,A -85,B 0,C 180,E1 -1435.884,E2 -1435.884} C_VEL
LIN {X 0,Y 587.158,Z 427.658,A -85,B 0,C 180,E1 -1436.915,E2 -1436.915} C_VEL
LIN {X 0,Y 587.137,Z 430.599,A -85,B 0,C 180,E1 -1437.944,E2 -1437.944} C_VEL
LIN {X 0,Y 587.147,Z 431.898,A -85,B 0,C 180,E1 -1438.63,E2 -1438.63} C_VEL
LIN {X 0,Y 587.136,Z 432.708,A -85,B 0,C 180,E1 -1439.316,E2 -1439.316} C_VEL
LIN {X 0,Y 587.135,Z 432.967,A -85,B 0,C 180,E1 -1440.002,E2 -1440.002} C_VEL
LIN {X 0,Y 587.139,Z 432.758,A -85,B 0,C 180,E1 -1440.688,E2 -1440.688} C_VEL
LIN {X 0,Y 587.146,Z 432.016,A -85,B 0,C 180,E1 -1441.374,E2 -1441.374} C_VEL
LIN {X 0,Y 587.14,Z 430.799,A -85,B 0,C 180,E1 -1442.06,E2 -1442.06} C_VEL
LIN {X 0,Y 587.157,Z 427.945,A -85,B 0,C 180,E1 -1443.09,E2 -1443.09} C_VEL
LIN {X 0,Y 587.209,Z 425.342,A -85,B 0,C 180,E1 -1443.776,E2 -1443.776} C_VEL
LIN {X 0,Y 587.171,Z 420.224,A -85,B 0,C 180,E1 -1444.808,E2 -1444.808} C_VEL
LIN {X 0,Y 587.239,Z 414.716,A -85,B 0,C 180,E1 -1445.668,E2 -1445.668} C_VEL
LIN {X 0,Y 587.271,Z 406.761,A -85,B 0,C 180,E1 -1446.645,E2 -1446.645} C_VEL
LIN {X 0,Y 587.312,Z 397.932,A -85,B 0,C 180,E1 -1447.479,E2 -1447.479} C_VEL
LIN {X 0,Y 587.349,Z 388.691,A -85,B 0,C 180,E1 -1448.171,E2 -1448.171} C_VEL
LIN {X 0,Y 587.4,Z 378.185,A -85,B 0,C 180,E1 -1448.777,E2 -1448.777} C_VEL
LIN {X 0,Y 587.455,Z 368.18,A -85,B 0,C 180,E1 -1449.209,E2 -1449.209} C_VEL
LIN {X 0,Y 587.497,Z 357.685,A -85,B 0,C 180,E1 -1449.534,E2 -1449.534} C_VEL
LIN {X 0,Y 587.558,Z 346.539,A -85,B 0,C 180,E1 -1449.751,E2 -1449.751} C_VEL
LIN {X 0,Y 587.418,Z 276.343,A -85,B 0,C 180,E1 -1450.61,E2 -1450.61} C_VEL
LIN {X 0,Y 587.221,Z 274.889,A -85,B 0,C 180,E1 -1450.643,E2 -1450.643} C_VEL
LIN {X 0,Y 587.276,Z 261.857,A -85,B 0,C 180,E1 -1453.497,E2 -1453.497} C_VEL
LIN {X 0,Y 587.331,Z 249.05,A -85,B 0,C 180,E1 -1456.334,E2 -1456.334} C_VEL
LIN {X 0,Y 587.379,Z 247.128,A -85,B 0,C 180,E1 -1456.793,E2 -1456.793} C_VEL
LIN {X 0,Y 587.311,Z 247.136,A -85,B 0,C 180,E1 -1459.578,E2 -1459.578} C_VEL
LIN {X 0,Y 587.318,Z 247.135,A -85,B 0,C 180,E1 -1461.776,E2 -1461.776} C_VEL
LIN {X 0,Y 587.324,Z 247.136,A -85,B 0,C 180,E1 -1464.761,E2 -1464.761} C_VEL
LIN {X 0,Y 587.309,Z 247.135,A -85,B 0,C 180,E1 -1467.684,E2 -1467.684} C_VEL
LIN {X 0,Y 587.32,Z 247.139,A -85,B 0,C 180,E1 -1470.172,E2 -1470.172} C_VEL
LIN {X 0,Y 587.344,Z 247.137,A -85,B 0,C 180,E1 -1472.58,E2 -1472.58} C_VEL
LIN {X 0,Y 587.315,Z 247.135,A -85,B 0,C 180,E1 -1475.058,E2 -1475.058} C_VEL
LIN {X 0,Y 587.338,Z 247.131,A -85,B 0,C 180,E1 -1477.838,E2 -1477.838} C_VEL
LIN {X 0,Y 587.313,Z 247.139,A -85,B 0,C 180,E1 -1480.256,E2 -1480.256} C_VEL
LIN {X 0,Y 587.32,Z 247.134,A -85,B 0,C 180,E1 -1483.118,E2 -1483.118} C_VEL
LIN {X 0,Y 587.318,Z 247.135,A -85,B 0,C 180,E1 -1486.049,E2 -1486.049} C_VEL
LIN {X 0,Y 587.339,Z 247.135,A -85,B 0,C 180,E1 -1488.926,E2 -1488.926} C_VEL
LIN {X 0,Y 587.322,Z 247.132,A -85,B 0,C 180,E1 -1491.52,E2 -1491.52} C_VEL
LIN {X 0,Y 587.293,Z 247.137,A -85,B 0,C 180,E1 -1494.1,E2 -1494.1} C_VEL
LIN {X 0,Y 587.342,Z 247.137,A -85,B 0,C 180,E1 -1496.889,E2 -1496.889} C_VEL
LIN {X 0,Y 587.326,Z 247.132,A -85,B 0,C 180,E1 -1499.493,E2 -1499.493} C_VEL
LIN {X 0,Y 587.346,Z 247.133,A -85,B 0,C 180,E1 -1502.309,E2 -1502.309} C_VEL
LIN {X 0,Y 587.351,Z 247.132,A -85,B 0,C 180,E1 -1505.241,E2 -1505.241} C_VEL
LIN {X 0,Y 587.35,Z 247.192,A -85,B 0,C 180,E1 -1507.672,E2 -1507.672} C_VEL
LIN {X 0,Y 587.709,Z 251.8,A -85,B 0,C 180,E1 -1508.425,E2 -1508.425} C_VEL
LIN {X 0,Y 587.576,Z 269.074,A -85,B 0,C 180,E1 -1511.159,E2 -1511.159} C_VEL
LIN {X 0,Y 587.424,Z 288.653,A -85,B 0,C 180,E1 -1514.206,E2 -1514.206} C_VEL
LIN {X 0,Y 587.36,Z 305.929,A -85,B 0,C 180,E1 -1516.859,E2 -1516.859} C_VEL
LIN {X 0,Y 587.293,Z 322.505,A -85,B 0,C 180,E1 -1519.379,E2 -1519.379} C_VEL
LIN {X 0,Y 587.591,Z 329.039,A -85,B 0,C 180,E1 -1519.471,E2 -1519.471} C_VEL
LIN {X 0,Y 587.499,Z 400.429,A -85,B 0,C 180,E1 -1520.359,E2 -1520.359} C_VEL
LIN {X 0,Y 587.45,Z 410.898,A -85,B 0,C 180,E1 -1520.597,E2 -1520.597} C_VEL
LIN {X 0,Y 587.413,Z 421.61,A -85,B 0,C 180,E1 -1520.965,E2 -1520.965} C_VEL
LIN {X 0,Y 587.392,Z 432.232,A -85,B 0,C 180,E1 -1521.485,E2 -1521.485} C_VEL
LIN {X 0,Y 587.344,Z 440.545,A -85,B 0,C 180,E1 -1522.004,E2 -1522.004} C_VEL
LIN {X 0,Y 587.293,Z 448.401,A -85,B 0,C 180,E1 -1522.609,E2 -1522.609} C_VEL
LIN {X 0,Y 587.295,Z 456.084,A -85,B 0,C 180,E1 -1523.334,E2 -1523.334} C_VEL
LIN {X 0,Y 587.253,Z 463.189,A -85,B 0,C 180,E1 -1524.161,E2 -1524.161} C_VEL
LIN {X 0,Y 587.17,Z 469.986,A -85,B 0,C 180,E1 -1525.194,E2 -1525.194} C_VEL
LIN {X 0,Y 587.211,Z 475.147,A -85,B 0,C 180,E1 -1526.226,E2 -1526.226} C_VEL
LIN {X 0,Y 587.155,Z 477.788,A -85,B 0,C 180,E1 -1526.912,E2 -1526.912} C_VEL
LIN {X 0,Y 587.141,Z 480.68,A -85,B 0,C 180,E1 -1527.942,E2 -1527.942} C_VEL
LIN {X 0,Y 587.145,Z 481.936,A -85,B 0,C 180,E1 -1528.628,E2 -1528.628} C_VEL
LIN {X 0,Y 587.136,Z 482.711,A -85,B 0,C 180,E1 -1529.314,E2 -1529.314} C_VEL
LIN {X 0,Y 587.134,Z 483,A -85,B 0,C 180,E1 -1530,E2 -1530} C_VEL
LIN {X 0,Y 587.136,Z 482.712,A -85,B 0,C 180,E1 -1530.686,E2 -1530.686} C_VEL
LIN {X 0,Y 587.145,Z 481.936,A -85,B 0,C 180,E1 -1531.372,E2 -1531.372} C_VEL
LIN {X 0,Y 587.141,Z 480.68,A -85,B 0,C 180,E1 -1532.058,E2 -1532.058} C_VEL
LIN {X 0,Y 587.155,Z 477.788,A -85,B 0,C 180,E1 -1533.087,E2 -1533.087} C_VEL
LIN {X 0,Y 587.211,Z 475.148,A -85,B 0,C 180,E1 -1533.774,E2 -1533.774} C_VEL
LIN {X 0,Y 587.17,Z 469.986,A -85,B 0,C 180,E1 -1534.806,E2 -1534.806} C_VEL
LIN {X 0,Y 587.253,Z 463.189,A -85,B 0,C 180,E1 -1535.838,E2 -1535.838} C_VEL
LIN {X 0,Y 587.27,Z 456.292,A -85,B 0,C 180,E1 -1536.645,E2 -1536.645} C_VEL
LIN {X 0,Y 587.292,Z 448.407,A -85,B 0,C 180,E1 -1537.391,E2 -1537.391} C_VEL
LIN {X 0,Y 587.34,Z 440.551,A -85,B 0,C 180,E1 -1537.996,E2 -1537.996} C_VEL
LIN {X 0,Y 587.411,Z 430.736,A -85,B 0,C 180,E1 -1538.601,E2 -1538.601} C_VEL
LIN {X 0,Y 587.427,Z 419.303,A -85,B 0,C 180,E1 -1539.121,E2 -1539.121} C_VEL
LIN {X 0,Y 587.458,Z 409.25,A -85,B 0,C 180,E1 -1539.446,E2 -1539.446} C_VEL
LIN {X 0,Y 587.499,Z 400.451,A -85,B 0,C 180,E1 -1539.641,E2 -1539.641} C_VEL
LIN {X 0,Y 587.598,Z 328.886,A -85,B 0,C 180,E1 -1540.531,E2 -1540.531} C_VEL
LIN {X 0,Y 587.293,Z 322.487,A -85,B 0,C 180,E1 -1540.624,E2 -1540.624} C_VEL
LIN {X 0,Y 587.388,Z 304.779,A -85,B 0,C 180,E1 -1543.316,E2 -1543.316} C_VEL
LIN {X 0,Y 587.475,Z 285.2,A -85,B 0,C 180,E1 -1546.328,E2 -1546.328} C_VEL
LIN {X 0,Y 587.574,Z 267.405,A -85,B 0,C 180,E1 -1549.104,E2 -1549.104} C_VEL
LIN {X 0,Y 587.704,Z 250.649,A -85,B 0,C 180,E1 -1551.759,E2 -1551.759} C_VEL
LIN {X 0,Y 587.341,Z 247.135,A -85,B 0,C 180,E1 -1552.375,E2 -1552.375} C_VEL
LIN {X 0,Y 587.352,Z 247.132,A -85,B 0,C 180,E1 -1554.758,E2 -1554.758} C_VEL
LIN {X 0,Y 587.345,Z 247.133,A -85,B 0,C 180,E1 -1557.691,E2 -1557.691} C_VEL
LIN {X 0,Y 587.328,Z 247.131,A -85,B 0,C 180,E1 -1560.508,E2 -1560.508} C_VEL
LIN {X 0,Y 587.341,Z 247.136,A -85,B 0,C 180,E1 -1563.111,E2 -1563.111} C_VEL
LIN {X 0,Y 587.292,Z 247.137,A -85,B 0,C 180,E1 -1565.9,E2 -1565.9} C_VEL
LIN {X 0,Y 587.322,Z 247.132,A -85,B 0,C 180,E1 -1568.48,E2 -1568.48} C_VEL
LIN {X 0,Y 587.338,Z 247.136,A -85,B 0,C 180,E1 -1571.157,E2 -1571.157} C_VEL
LIN {X 0,Y 587.316,Z 247.134,A -85,B 0,C 180,E1 -1574.111,E2 -1574.111} C_VEL
LIN {X 0,Y 587.319,Z 247.135,A -85,B 0,C 180,E1 -1576.993,E2 -1576.993} C_VEL
LIN {X 0,Y 587.313,Z 247.14,A -85,B 0,C 180,E1 -1579.744,E2 -1579.744} C_VEL
LIN {X 0,Y 587.346,Z 247.129,A -85,B 0,C 180,E1 -1582.391,E2 -1582.391} C_VEL
LIN {X 0,Y 587.345,Z 247.14,A -85,B 0,C 180,E1 -1585.653,E2 -1585.653} C_VEL
LIN {X 0,Y 587.343,Z 247.131,A -85,B 0,C 180,E1 -1588.23,E2 -1588.23} C_VEL
LIN {X 0,Y 587.349,Z 247.128,A -85,B 0,C 180,E1 -1590.867,E2 -1590.867} C_VEL
LIN {X 0,Y 587.337,Z 247.139,A -85,B 0,C 180,E1 -1593.824,E2 -1593.824} C_VEL
LIN {X 0,Y 587.321,Z 247.139,A -85,B 0,C 180,E1 -1595.991,E2 -1595.991} C_VEL
LIN {X 0,Y 587.321,Z 247.135,A -85,B 0,C 180,E1 -1598.224,E2 -1598.224} C_VEL
LIN {X 0,Y 587.35,Z 247.129,A -85,B 0,C 180,E1 -1601.15,E2 -1601.15} C_VEL
LIN {X 0,Y 587.32,Z 247.14,A -85,B 0,C 180,E1 -1604.023,E2 -1604.023} C_VEL
LIN {X 0,Y 587.355,Z 247.134,A -85,B 0,C 180,E1 -1606.152,E2 -1606.152} C_VEL
LIN {X 0,Y 587.343,Z 247.128,A -85,B 0,C 180,E1 -1608.961,E2 -1608.961} C_VEL
LIN {X 0,Y 587.367,Z 247.132,A -85,B 0,C 180,E1 -1611.743,E2 -1611.743} C_VEL
LIN {X 0,Y 587.341,Z 247.131,A -85,B 0,C 180,E1 -1614.505,E2 -1614.505} C_VEL
LIN {X 0,Y 587.369,Z 247.126,A -85,B 0,C 180,E1 -1617.255,E2 -1617.255} C_VEL
LIN {X 0,Y 587.385,Z 247.132,A -85,B 0,C 180,E1 -1619.998,E2 -1619.998} C_VEL
LIN {X 0,Y 587.356,Z 247.129,A -85,B 0,C 180,E1 -1622.741,E2 -1622.741} C_VEL
LIN {X 0,Y 587.345,Z 247.129,A -85,B 0,C 180,E1 -1625.491,E2 -1625.491} C_VEL
LIN {X 0,Y 587.361,Z 247.137,A -85,B 0,C 180,E1 -1628.253,E2 -1628.253} C_VEL
LIN {X 0,Y 587.344,Z 247.128,A -85,B 0,C 180,E1 -1631.131,E2 -1631.131} C_VEL
LIN {X 0,Y 587.359,Z 247.138,A -85,B 0,C 180,E1 -1634.258,E2 -1634.258} C_VEL
LIN {X 0,Y 587.334,Z 247.13,A -85,B 0,C 180,E1 -1637.403,E2 -1637.403} C_VEL
LIN {X 0,Y 587.3,Z 247.139,A -85,B 0,C 180,E1 -1638.291,E2 -1638.291} C_VEL
LIN {X 0,Y 586.654,Z 247.218,A -85,B 0,C 180,E1 -1638.863,E2 -1638.863} C_VEL
LIN {X 0,Y 583.831,Z 247.568,A -85,B 0,C 180,E1 -1639.792,E2 -1639.792} C_VEL
LIN {X 0,Y 581.423,Z 247.874,A -85,B 0,C 180,E1 -1640.539,E2 -1640.539} C_VEL
LIN {X 0,Y 580.37,Z 247.999,A -85,B 0,C 180,E1 -1641.115,E2 -1641.115} C_VEL
LIN {X 0,Y 580.274,Z 248.009,A -85,B 0,C 180,E1 -1641.31,E2 -1641.31} C_VEL
LIN {X 0,Y 580.287,Z 248.017,A -85,B 0,C 180,E1 -1644.313,E2 -1644.313} C_VEL
LIN {X 0,Y 580.263,Z 248.019,A -85,B 0,C 180,E1 -1646.621,E2 -1646.621} C_VEL
LIN {X 0,Y 580.29,Z 248.008,A -85,B 0,C 180,E1 -1649.308,E2 -1649.308} C_VEL
LIN {X 0,Y 580.284,Z 248.013,A -85,B 0,C 180,E1 -1652.197,E2 -1652.197} C_VEL
LIN {X 0,Y 580.274,Z 248.017,A -85,B 0,C 180,E1 -1654.693,E2 -1654.693} C_VEL
LIN {X 0,Y 580.28,Z 248.01,A -85,B 0,C 180,E1 -1657.265,E2 -1657.265} C_VEL
LIN {X 0,Y 580.279,Z 248.013,A -85,B 0,C 180,E1 -1660.269,E2 -1660.269} C_VEL
LIN {X 0,Y 580.272,Z 248.02,A -85,B 0,C 180,E1 -1662.702,E2 -1662.702} C_VEL
LIN {X 0,Y 580.248,Z 248.013,A -85,B 0,C 180,E1 -1665.606,E2 -1665.606} C_VEL
LIN {X 0,Y 580.277,Z 248.019,A -85,B 0,C 180,E1 -1668.663,E2 -1668.663} C_VEL
LIN {X 0,Y 580.266,Z 248.019,A -85,B 0,C 180,E1 -1670.964,E2 -1670.964} C_VEL
LIN {X 0,Y 580.267,Z 248.012,A -85,B 0,C 180,E1 -1673.596,E2 -1673.596} C_VEL
LIN {X 0,Y 580.31,Z 248.065,A -85,B 0,C 180,E1 -1676.331,E2 -1676.331} C_VEL
LIN {X 0,Y 580.164,Z 259.928,A -85,B 0,C 180,E1 -1678.995,E2 -1678.995} C_VEL
LIN {X 0,Y 580.161,Z 270.802,A -85,B 0,C 180,E1 -1681.413,E2 -1681.413} C_VEL
LIN {X 0,Y 580.192,Z 274.916,A -85,B 0,C 180,E1 -1682.323,E2 -1682.323} C_VEL
LIN {X 0,Y 580.601,Z 279.896,A -85,B 0,C 180,E1 -1682.398,E2 -1682.398} C_VEL
LIN {X 0,Y 580.514,Z 349.282,A -85,B 0,C 180,E1 -1683.267,E2 -1683.267} C_VEL
LIN {X 0,Y 580.461,Z 358.533,A -85,B 0,C 180,E1 -1683.465,E2 -1683.465} C_VEL
LIN {X 0,Y 580.449,Z 366.222,A -85,B 0,C 180,E1 -1683.701,E2 -1683.701} C_VEL
LIN {X 0,Y 580.411,Z 375.448,A -85,B 0,C 180,E1 -1684.078,E2 -1684.078} C_VEL
LIN {X 0,Y 580.355,Z 384.157,A -85,B 0,C 180,E1 -1684.539,E2 -1684.539} C_VEL
LIN {X 0,Y 580.308,Z 393.075,A -85,B 0,C 180,E1 -1685.133,E2 -1685.133} C_VEL
LIN {X 0,Y 580.239,Z 401.916,A -85,B 0,C 180,E1 -1685.871,E2 -1685.871} C_VEL
LIN {X 0,Y 580.204,Z 408.832,A -85,B 0,C 180,E1 -1686.599,E2 -1686.599} C_VEL
LIN {X 0,Y 580.148,Z 414.907,A -85,B 0,C 180,E1 -1687.38,E2 -1687.38} C_VEL
LIN {X 0,Y 580.122,Z 419.701,A -85,B 0,C 180,E1 -1688.129,E2 -1688.129} C_VEL
LIN {X 0,Y 580.113,Z 423.607,A -85,B 0,C 180,E1 -1688.871,E2 -1688.871} C_VEL
LIN {X 0,Y 580.079,Z 427.393,A -85,B 0,C 180,E1 -1689.8,E2 -1689.8} C_VEL
LIN {X 0,Y 580.056,Z 430.55,A -85,B 0,C 180,E1 -1690.905,E2 -1690.905} C_VEL
LIN {X 0,Y 580.022,Z 431.909,A -85,B 0,C 180,E1 -1691.637,E2 -1691.637} C_VEL
LIN {X 0,Y 580.027,Z 432.718,A -85,B 0,C 180,E1 -1692.367,E2 -1692.367} C_VEL
LIN {X 0,Y 580.067,Z 432.977,A -85,B 0,C 180,E1 -1693.152,E2 -1693.152} C_VEL
LIN {X 0,Y 580.053,Z 432.673,A -85,B 0,C 180,E1 -1693.819,E2 -1693.819} C_VEL
LIN {X 0,Y 580.05,Z 431.787,A -85,B 0,C 180,E1 -1694.541,E2 -1694.541} C_VEL
LIN {X 0,Y 580.091,Z 429.226,A -85,B 0,C 180,E1 -1695.732,E2 -1695.732} C_VEL
LIN {X 0,Y 580.079,Z 425.907,A -85,B 0,C 180,E1 -1696.691,E2 -1696.691} C_VEL
LIN {X 0,Y 580.096,Z 422.751,A -85,B 0,C 180,E1 -1697.404,E2 -1697.404} C_VEL
LIN {X 0,Y 580.157,Z 417.72,A -85,B 0,C 180,E1 -1698.293,E2 -1698.293} C_VEL
LIN {X 0,Y 580.178,Z 412.963,A -85,B 0,C 180,E1 -1698.984,E2 -1698.984} C_VEL
LIN {X 0,Y 580.204,Z 406.905,A -85,B 0,C 180,E1 -1699.708,E2 -1699.708} C_VEL
LIN {X 0,Y 580.238,Z 399.716,A -85,B 0,C 180,E1 -1700.413,E2 -1700.413} C_VEL
LIN {X 0,Y 580.3,Z 392.067,A -85,B 0,C 180,E1 -1701.029,E2 -1701.029} C_VEL
LIN {X 0,Y 580.317,Z 384.078,A -85,B 0,C 180,E1 -1701.556,E2 -1701.556} C_VEL
LIN {X 0,Y 580.384,Z 375.805,A -85,B 0,C 180,E1 -1701.995,E2 -1701.995} C_VEL
LIN {X 0,Y 580.403,Z 367.433,A -85,B 0,C 180,E1 -1702.346,E2 -1702.346} C_VEL
LIN {X 0,Y 580.479,Z 358.13,A -85,B 0,C 180,E1 -1702.635,E2 -1702.635} C_VEL
LIN {X 0,Y 580.525,Z 348.819,A -85,B 0,C 180,E1 -1702.831,E2 -1702.831} C_VEL
LIN {X 0,Y 580.561,Z 277.926,A -85,B 0,C 180,E1 -1703.717,E2 -1703.717} C_VEL
LIN {X 0,Y 580.154,Z 274.841,A -85,B 0,C 180,E1 -1703.785,E2 -1703.785} C_VEL
LIN {X 0,Y 580.207,Z 264.027,A -85,B 0,C 180,E1 -1706.18,E2 -1706.18} C_VEL
LIN {X 0,Y 580.271,Z 251.611,A -85,B 0,C 180,E1 -1708.959,E2 -1708.959} C_VEL
LIN {X 0,Y 580.296,Z 248.01,A -85,B 0,C 180,E1 -1709.783,E2 -1709.783} C_VEL
LIN {X 0,Y 580.306,Z 248.009,A -85,B 0,C 180,E1 -1712.777,E2 -1712.777} C_VEL
LIN {X 0,Y 580.3,Z 248.012,A -85,B 0,C 180,E1 -1715.56,E2 -1715.56} C_VEL
LIN {X 0,Y 580.271,Z 248.01,A -85,B 0,C 180,E1 -1718.357,E2 -1718.357} C_VEL
LIN {X 0,Y 580.299,Z 248.015,A -85,B 0,C 180,E1 -1721.212,E2 -1721.212} C_VEL
LIN {X 0,Y 580.253,Z 248.012,A -85,B 0,C 180,E1 -1724.331,E2 -1724.331} C_VEL
LIN {X 0,Y 580.273,Z 248.013,A -85,B 0,C 180,E1 -1726.915,E2 -1726.915} C_VEL
LIN {X 0,Y 580.262,Z 248.015,A -85,B 0,C 180,E1 -1729.824,E2 -1729.824} C_VEL
LIN {X 0,Y 580.23,Z 248.017,A -85,B 0,C 180,E1 -1732.055,E2 -1732.055} C_VEL
LIN {X 0,Y 580.253,Z 248.017,A -85,B 0,C 180,E1 -1735.082,E2 -1735.082} C_VEL
LIN {X 0,Y 580.252,Z 248.013,A -85,B 0,C 180,E1 -1738.188,E2 -1738.188} C_VEL
LIN {X 0,Y 580.238,Z 248.014,A -85,B 0,C 180,E1 -1740.695,E2 -1740.695} C_VEL
LIN {X 0,Y 580.273,Z 248.017,A -85,B 0,C 180,E1 -1743.319,E2 -1743.319} C_VEL
LIN {X 0,Y 580.212,Z 248.024,A -85,B 0,C 180,E1 -1745.758,E2 -1745.758} C_VEL
LIN {X 0,Y 580.252,Z 248.014,A -85,B 0,C 180,E1 -1748.149,E2 -1748.149} C_VEL
LIN {X 0,Y 580.265,Z 248.012,A -85,B 0,C 180,E1 -1750.847,E2 -1750.847} C_VEL
LIN {X 0,Y 580.242,Z 248.024,A -85,B 0,C 180,E1 -1753.662,E2 -1753.662} C_VEL
LIN {X 0,Y 580.243,Z 248.014,A -85,B 0,C 180,E1 -1756.613,E2 -1756.613} C_VEL
LIN {X 0,Y 580.275,Z 248.013,A -85,B 0,C 180,E1 -1759.159,E2 -1759.159} C_VEL
LIN {X 0,Y 580.264,Z 248.017,A -85,B 0,C 180,E1 -1761.931,E2 -1761.931} C_VEL
LIN {X 0,Y 580.258,Z 248.012,A -85,B 0,C 180,E1 -1764.457,E2 -1764.457} C_VEL
LIN {X 0,Y 580.27,Z 248.011,A -85,B 0,C 180,E1 -1766.978,E2 -1766.978} C_VEL
LIN {X 0,Y 580.278,Z 248.015,A -85,B 0,C 180,E1 -1769.428,E2 -1769.428} C_VEL
LIN {X 0,Y 580.243,Z 248.018,A -85,B 0,C 180,E1 -1772.152,E2 -1772.152} C_VEL
LIN {X 0,Y 580.309,Z 248.008,A -85,B 0,C 180,E1 -1775.273,E2 -1775.273} C_VEL
LIN {X 0,Y 580.257,Z 248.02,A -85,B 0,C 180,E1 -1777.95,E2 -1777.95} C_VEL
LIN {X 0,Y 580.277,Z 248.01,A -85,B 0,C 180,E1 -1780.916,E2 -1780.916} C_VEL
LIN {X 0,Y 580.28,Z 248.103,A -85,B 0,C 180,E1 -1783.339,E2 -1783.339} C_VEL
LIN {X 0,Y 580.232,Z 261.471,A -85,B 0,C 180,E1 -1786.341,E2 -1786.341} C_VEL
LIN {X 0,Y 580.131,Z 274.539,A -85,B 0,C 180,E1 -1789.238,E2 -1789.238} C_VEL
LIN {X 0,Y 580.144,Z 275.128,A -85,B 0,C 180,E1 -1789.331,E2 -1789.331} C_VEL
LIN {X 0,Y 580.594,Z 281.093,A -85,B 0,C 180,E1 -1789.413,E2 -1789.413} C_VEL
LIN {X 0,Y 580.527,Z 350.67,A -85,B 0,C 180,E1 -1790.289,E2 -1790.289} C_VEL
LIN {X 0,Y 580.464,Z 361.838,A -85,B 0,C 180,E1 -1790.551,E2 -1790.551} C_VEL
LIN {X 0,Y 580.386,Z 372.645,A -85,B 0,C 180,E1 -1790.945,E2 -1790.945} C_VEL
LIN {X 0,Y 580.347,Z 383.079,A -85,B 0,C 180,E1 -1791.471,E2 -1791.471} C_VEL
LIN {X 0,Y 580.289,Z 393.641,A -85,B 0,C 180,E1 -1792.172,E2 -1792.172} C_VEL
LIN {X 0,Y 580.245,Z 401.856,A -85,B 0,C 180,E1 -1792.871,E2 -1792.871} C_VEL
LIN {X 0,Y 580.196,Z 408.67,A -85,B 0,C 180,E1 -1793.583,E2 -1793.583} C_VEL
LIN {X 0,Y 580.174,Z 414.124,A -85,B 0,C 180,E1 -1794.267,E2 -1794.267} C_VEL
LIN {X 0,Y 580.1,Z 419.748,A -85,B 0,C 180,E1 -1795.138,E2 -1795.138} C_VEL
LIN {X 0,Y 580.105,Z 423.455,A -85,B 0,C 180,E1 -1795.834,E2 -1795.834} C_VEL
LIN {X 0,Y 580.072,Z 427.665,A -85,B 0,C 180,E1 -1796.877,E2 -1796.877} C_VEL
LIN {X 0,Y 580.037,Z 430.606,A -85,B 0,C 180,E1 -1797.919,E2 -1797.919} C_VEL
LIN {X 0,Y 580.047,Z 431.906,A -85,B 0,C 180,E1 -1798.614,E2 -1798.614} C_VEL
LIN {X 0,Y 580.036,Z 432.705,A -85,B 0,C 180,E1 -1799.308,E2 -1799.308} C_VEL
LIN {X 0,Y 580.036,Z 432.957,A -85,B 0,C 180,E1 -1800.002,E2 -1800.002} C_VEL
LIN {X 0,Y 580.039,Z 432.765,A -85,B 0,C 180,E1 -1800.696,E2 -1800.696} C_VEL
LIN {X 0,Y 580.046,Z 432.023,A -85,B 0,C 180,E1 -1801.391,E2 -1801.391} C_VEL
LIN {X 0,Y 580.04,Z 430.798,A -85,B 0,C 180,E1 -1802.085,E2 -1802.085} C_VEL
LIN {X 0,Y 580.072,Z 427.948,A -85,B 0,C 180,E1 -1803.127,E2 -1803.127} C_VEL
LIN {X 0,Y 580.122,Z 425.335,A -85,B 0,C 180,E1 -1803.823,E2 -1803.823} C_VEL
LIN {X 0,Y 580.077,Z 420.221,A -85,B 0,C 180,E1 -1804.867,E2 -1804.867} C_VEL
LIN {X 0,Y 580.174,Z 414.709,A -85,B 0,C 180,E1 -1805.738,E2 -1805.738} C_VEL
LIN {X 0,Y 580.198,Z 407.491,A -85,B 0,C 180,E1 -1806.647,E2 -1806.647} C_VEL
LIN {X 0,Y 580.254,Z 398.951,A -85,B 0,C 180,E1 -1807.483,E2 -1807.483} C_VEL
LIN {X 0,Y 580.295,Z 389.984,A -85,B 0,C 180,E1 -1808.183,E2 -1808.183} C_VEL
LIN {X 0,Y 580.389,Z 379.84,A -85,B 0,C 180,E1 -1808.796,E2 -1808.796} C_VEL
LIN {X 0,Y 580.461,Z 369.38,A -85,B 0,C 180,E1 -1809.277,E2 -1809.277} C_VEL
LIN {X 0,Y 580.486,Z 357.694,A -85,B 0,C 180,E1 -1809.651,E2 -1809.651} C_VEL
LIN {X 0,Y 580.586,Z 346.505,A -85,B 0,C 180,E1 -1809.869,E2 -1809.869} C_VEL
LIN {X 0,Y 580.431,Z 277.042,A -85,B 0,C 180,E1 -1810.73,E2 -1810.73} C_VEL
LIN {X 0,Y 580.165,Z 274.892,A -85,B 0,C 180,E1 -1810.773,E2 -1810.773} C_VEL
LIN {X 0,Y 580.2,Z 261.854,A -85,B 0,C 180,E1 -1813.664,E2 -1813.664} C_VEL
LIN {X 0,Y 580.301,Z 249.047,A -85,B 0,C 180,E1 -1816.537,E2 -1816.537} C_VEL
LIN {X 0,Y 580.331,Z 248.006,A -85,B 0,C 180,E1 -1816.819,E2 -1816.819} C_VEL
LIN {X 0,Y 580.288,Z 248.013,A -85,B 0,C 180,E1 -1819.825,E2 -1819.825} C_VEL
LIN {X 0,Y 580.27,Z 248.017,A -85,B 0,C 180,E1 -1822.054,E2 -1822.054} C_VEL
LIN {X 0,Y 580.289,Z 248.009,A -85,B 0,C 180,E1 -1825.082,E2 -1825.082} C_VEL
LIN {X 0,Y 580.287,Z 248.016,A -85,B 0,C 180,E1 -1828.188,E2 -1828.188} C_VEL
LIN {X 0,Y 580.278,Z 248.015,A -85,B 0,C 180,E1 -1830.693,E2 -1830.693} C_VEL
LIN {X 0,Y 580.288,Z 248.009,A -85,B 0,C 180,E1 -1833.313,E2 -1833.313} C_VEL
LIN {X 0,Y 580.238,Z 248.015,A -85,B 0,C 180,E1 -1835.755,E2 -1835.755} C_VEL
LIN {X 0,Y 580.29,Z 248.013,A -85,B 0,C 180,E1 -1838.147,E2 -1838.147} C_VEL
LIN {X 0,Y 580.3,Z 248.012,A -85,B 0,C 180,E1 -1840.844,E2 -1840.844} C_VEL
LIN {X 0,Y 580.279,Z 248.009,A -85,B 0,C 180,E1 -1843.659,E2 -1843.659} C_VEL
LIN {X 0,Y 580.274,Z 248.02,A -85,B 0,C 180,E1 -1846.611,E2 -1846.611} C_VEL
LIN {X 0,Y 580.301,Z 248.009,A -85,B 0,C 180,E1 -1849.156,E2 -1849.156} C_VEL
LIN {X 0,Y 580.29,Z 248.009,A -85,B 0,C 180,E1 -1851.928,E2 -1851.928} C_VEL
LIN {X 0,Y 580.254,Z 248.019,A -85,B 0,C 180,E1 -1854.453,E2 -1854.453} C_VEL
LIN {X 0,Y 580.293,Z 248.013,A -85,B 0,C 180,E1 -1856.975,E2 -1856.975} C_VEL
LIN {X 0,Y 580.287,Z 248.009,A -85,B 0,C 180,E1 -1859.424,E2 -1859.424} C_VEL
LIN {X 0,Y 580.296,Z 248.009,A -85,B 0,C 180,E1 -1862.143,E2 -1862.143} C_VEL
LIN {X 0,Y 580.324,Z 248.008,A -85,B 0,C 180,E1 -1865.27,E2 -1865.27} C_VEL
LIN {X 0,Y 580.325,Z 248.162,A -85,B 0,C 180,E1 -1867.574,E2 -1867.574} C_VEL
LIN {X 0,Y 580.748,Z 252.906,A -85,B 0,C 180,E1 -1868.34,E2 -1868.34} C_VEL
LIN {X 0,Y 580.613,Z 269.074,A -85,B 0,C 180,E1 -1870.924,E2 -1870.924} C_VEL
LIN {X 0,Y 580.43,Z 287.502,A -85,B 0,C 180,E1 -1873.83,E2 -1873.83} C_VEL
LIN {X 0,Y 580.334,Z 305.929,A -85,B 0,C 180,E1 -1876.697,E2 -1876.697} C_VEL
LIN {X 0,Y 580.216,Z 322.471,A -85,B 0,C 180,E1 -1879.243,E2 -1879.243} C_VEL
LIN {X 0,Y 580.637,Z 329.347,A -85,B 0,C 180,E1 -1879.347,E2 -1879.347} C_VEL
LIN {X 0,Y 580.521,Z 400.428,A -85,B 0,C 180,E1 -1880.242,E2 -1880.242} C_VEL
LIN {X 0,Y 580.462,Z 410.898,A -85,B 0,C 180,E1 -1880.483,E2 -1880.483} C_VEL
LIN {X 0,Y 580.414,Z 421.608,A -85,B 0,C 180,E1 -1880.855,E2 -1880.855} C_VEL
LIN {X 0,Y 580.37,Z 432.229,A -85,B 0,C 180,E1 -1881.381,E2 -1881.381} C_VEL
LIN {X 0,Y 580.302,Z 440.542,A -85,B 0,C 180,E1 -1881.906,E2 -1881.906} C_VEL
LIN {X 0,Y 580.251,Z 448.401,A -85,B 0,C 180,E1 -1882.518,E2 -1882.518} C_VEL
LIN {X 0,Y 580.228,Z 455.467,A -85,B 0,C 180,E1 -1883.189,E2 -1883.189} C_VEL
LIN {X 0,Y 580.193,Z 463.189,A -85,B 0,C 180,E1 -1884.09,E2 -1884.09} C_VEL
LIN {X 0,Y 580.084,Z 469.986,A -85,B 0,C 180,E1 -1885.135,E2 -1885.135} C_VEL
LIN {X 0,Y 580.123,Z 475.147,A -85,B 0,C 180,E1 -1886.179,E2 -1886.179} C_VEL
LIN {X 0,Y 580.071,Z 477.788,A -85,B 0,C 180,E1 -1886.874,E2 -1886.874} C_VEL
LIN {X 0,Y 580.04,Z 480.681,A -85,B 0,C 180,E1 -1887.917,E2 -1887.917} C_VEL
LIN {X 0,Y 580.045,Z 481.936,A -85,B 0,C 180,E1 -1888.611,E2 -1888.611} C_VEL
LIN {X 0,Y 580.036,Z 482.711,A -85,B 0,C 180,E1 -1889.306,E2 -1889.306} C_VEL
LIN {X 0,Y 580.034,Z 483,A -85,B 0,C 180,E1 -1890,E2 -1890} C_VEL
LIN {X 0,Y 580.036,Z 482.711,A -85,B 0,C 180,E1 -1890.694,E2 -1890.694} C_VEL
LIN {X 0,Y 580.045,Z 481.936,A -85,B 0,C 180,E1 -1891.388,E2 -1891.388} C_VEL
LIN {X 0,Y 580.04,Z 480.681,A -85,B 0,C 180,E1 -1892.083,E2 -1892.083} C_VEL
LIN {X 0,Y 580.07,Z 477.788,A -85,B 0,C 180,E1 -1893.125,E2 -1893.125} C_VEL
LIN {X 0,Y 580.123,Z 475.148,A -85,B 0,C 180,E1 -1893.82,E2 -1893.82} C_VEL
LIN {X 0,Y 580.084,Z 469.986,A -85,B 0,C 180,E1 -1894.865,E2 -1894.865} C_VEL
LIN {X 0,Y 580.193,Z 463.188,A -85,B 0,C 180,E1 -1895.91,E2 -1895.91} C_VEL
LIN {X 0,Y 580.226,Z 455.501,A -85,B 0,C 180,E1 -1896.807,E2 -1896.807} C_VEL
LIN {X 0,Y 580.251,Z 448.408,A -85,B 0,C 180,E1 -1897.481,E2 -1897.481} C_VEL
LIN {X 0,Y 580.3,Z 440.548,A -85,B 0,C 180,E1 -1898.093,E2 -1898.093} C_VEL
LIN {X 0,Y 580.4,Z 430.734,A -85,B 0,C 180,E1 -1898.706,E2 -1898.706} C_VEL
LIN {X 0,Y 580.408,Z 419.305,A -85,B 0,C 180,E1 -1899.232,E2 -1899.232} C_VEL
LIN {X 0,Y 580.471,Z 409.25,A -85,B 0,C 180,E1 -1899.561,E2 -1899.561} C_VEL
LIN {X 0,Y 580.521,Z 400.45,A -85,B 0,C 180,E1 -1899.758,E2 -1899.758} C_VEL
LIN {X 0,Y 580.638,Z 328.849,A -85,B 0,C 180,E1 -1900.659,E2 -1900.659} C_VEL
LIN {X 0,Y 580.325,Z 323.403,A -85,B 0,C 180,E1 -1900.732,E2 -1900.732} C_VEL
LIN {X 0,Y 580.209,Z 322.54,A -85,B 0,C 180,E1 -1900.747,E2 -1900.747} C_VEL
LIN {X 0,Y 580.334,Z 305.931,A -85,B 0,C 180,E1 -1903.303,E2 -1903.303} C_VEL
LIN {X 0,Y 580.429,Z 287.504,A -85,B 0,C 180,E1 -1906.17,E2 -1906.17} C_VEL
LIN {X 0,Y 580.613,Z 269.076,A -85,B 0,C 180,E1 -1909.076,E2 -1909.076} C_VEL
LIN {X 0,Y 580.749,Z 251.719,A -85,B 0,C 180,E1 -1911.847,E2 -1911.847} C_VEL
LIN {X 0,Y 580.315,Z 248.011,A -85,B 0,C 180,E1 -1912.473,E2 -1912.473} C_VEL
LIN {X 0,Y 580.306,Z 248.015,A -85,B 0,C 180,E1 -1915.08,E2 -1915.08} C_VEL
LIN {X 0,Y 580.299,Z 248.007,A -85,B 0,C 180,E1 -1918.185,E2 -1918.185} C_VEL
LIN {X 0,Y 580.279,Z 248.011,A -85,B 0,C 180,E1 -1920.693,E2 -1920.693} C_VEL
LIN {X 0,Y 580.287,Z 248.018,A -85,B 0,C 180,E1 -1923.313,E2 -1923.313} C_VEL
LIN {X 0,Y 580.247,Z 248.017,A -85,B 0,C 180,E1 -1925.756,E2 -1925.756} C_VEL
LIN {X 0,Y 580.287,Z 248.009,A -85,B 0,C 180,E1 -1928.146,E2 -1928.146} C_VEL
LIN {X 0,Y 580.3,Z 248.008,A -85,B 0,C 180,E1 -1930.843,E2 -1930.843} C_VEL
